// TIA Portal V17 program export: 1 tag tables, 23 data types, 8 data blocks, 12 code blocks (in call order from the OBs), 7 instance data blocks

VAR_GLOBAL   // PLC tag table "默认变量表"
   Tag_1 AT %M0.2 : Bool;
   System_Byte AT %MB1 : Byte;
   FirstScan AT %M1.0 : Bool;
   DiagStatusUpdate AT %M1.1 : Bool;
   AlwaysTRUE AT %M1.2 : Bool;
   AlwaysFALSE AT %M1.3 : Bool;
   Clock_Byte AT %MB0 : Byte;
   Clock_10Hz AT %M0.0 : Bool;
   Clock_5Hz AT %M0.1 : Bool;
   "Clock_2.5Hz" AT %M0.2 : Bool;
   Clock_2Hz AT %M0.3 : Bool;
   "Clock_1.25Hz" AT %M0.4 : Bool;
   Clock_1Hz AT %M0.5 : Bool;
   "Clock_0.625Hz" AT %M0.6 : Bool;
   "Clock_0.5Hz" AT %M0.7 : Bool;
   "PositioningAxis_1_Actor_Interface_AddressIn(8)" AT %I256.0 : "PD_TEL105_IN";
   "PositioningAxis_1_Actor_Interface_AddressOut(8)" AT %Q256.0 : "PD_TEL105_OUT";
   profiSafeCtrl1 AT %Q276.0 : "LDrvSafe_typeSinaTlg901Control";
   proSafeStatus1 AT %I276.0 : "LDrvSafe_typeSinaTlg901Status";
   profiSafeCtrl2 AT %Q310.0 : "LDrvSafe_typeSinaSTlg30Control";
   profiSafeStatus2 AT %I310.0 : "LDrvSafe_typeSinaSTlg30Status";
   "PositioningAxis_2_Actor_Interface_AddressIn(7)" AT %I290.0 : "PD_TEL105_IN";
   "PositioningAxis_2_Actor_Interface_AddressOut(7)" AT %Q290.0 : "PD_TEL105_OUT";
END_VAR

TYPE "LDrvSafe_typeSinaSTlg30Control"
TITLE = LDrvSafe_typeSinaSTlg30Control
// Failsafe user-defined data type for PROFIsafe telegram 30 to control the Safety Integrated Functions of SINAMICS S
// stored: IsFailsafeCompliant true
   STRUCT
      STO { ExternalWritable := 'False'} : Bool;   // Safety Function Safe Torque Off
      SS1 { ExternalWritable := 'False'} : Bool;   // Safety Function Safe Stop 1
      SS2 { ExternalWritable := 'False'} : Bool;   // Safety Function Safe Stop 2
      SOS { ExternalWritable := 'False'} : Bool;   // Safety Function Safe Operating Stop
      SLS { ExternalWritable := 'False'} : Bool;   // Safety Function Safely-limited Speed
      reserved1 { ExternalWritable := 'False'} : Bool;   // Reserve bit 1
      SLP { ExternalWritable := 'False'} : Bool;   // Safety Function Safely-limited Position
      internalEventAcknowledge { ExternalWritable := 'False'} : Bool;   // Acknowledge Safety errors in the drive
      SLA { ExternalWritable := 'False'} : Bool;   // Safety Function Safely-limited Acceleration
      selectSLSbit0 { ExternalWritable := 'False'} : Bool;   // Select one of the the four SLS limits; operates together with bit 1
      selectSLSbit1 { ExternalWritable := 'False'} : Bool;   // Select one of the the four SLS limits; operates together with bit 0
      reserved3 { ExternalWritable := 'False'} : Bool;   // Reserve bit 3
      SDIpositive { ExternalWritable := 'False'} : Bool;   // Safety Function Safe Direction (positive direction)
      SDInegative { ExternalWritable := 'False'} : Bool;   // Safety Function Safe Direction (negative direction)
      reserved4 { ExternalWritable := 'False'} : Bool;   // Reserve bit 4
      reserved5 { ExternalWritable := 'False'} : Bool;   // Reserve bit 5
   END_STRUCT;
END_TYPE

TYPE "LDrvSafe_typeSinaSTlg30Status"
TITLE = LDrvSafe_typeSinaSTlg30Status
// Failsafe user-defined data type for PROFIsafe telegram 30 to get status information of Safety Integrated Functions of SINAMICS S
// stored: IsFailsafeCompliant true
   STRUCT
      STOactive { ExternalWritable := 'False'} : Bool;   // Safety Function Safe Torque Off active
      SS1active { ExternalWritable := 'False'} : Bool;   // Safety Function Safe Stop 1 active
      SS2active { ExternalWritable := 'False'} : Bool;   // Safety Function Safe Stop 2 active
      SOSactive { ExternalWritable := 'False'} : Bool;   // Safety Function Safe Operating Stop active
      SLSactive { ExternalWritable := 'False'} : Bool;   // Safety Function Safely-limited Speed active
      reserved1 { ExternalWritable := 'False'} : Bool;   // Reserve bit 1
      SLPactive { ExternalWritable := 'False'} : Bool;   // Safety Function Safely-limited Position active
      internalEvent { ExternalWritable := 'False'} : Bool;   // Internal Event occured (Safety error in SINAMICS)
      SLAactive { ExternalWritable := 'False'} : Bool;   // Safety Function Safely-limited Acceleration active
      SLSbit0Active { ExternalWritable := 'False'} : Bool;   // One of the the four SLS limits is active; operates together with bit 1
      SLSbit1Active { ExternalWritable := 'False'} : Bool;   // One of the the four SLS limits is active; operates together with bit 0
      SOSselected { ExternalWritable := 'False'} : Bool;   // Safety Function Safe Operating Stop selected (not active yet)
      SDIpositiveActive { ExternalWritable := 'False'} : Bool;   // Safety Function Safe Direction (positive direction) active
      SDInegativeActive { ExternalWritable := 'False'} : Bool;   // Safety Function Safe Direction (negative direction) active
      reserved3 { ExternalWritable := 'False'} : Bool;   // Reserve bit 3
      SSMactive { ExternalWritable := 'False'} : Bool;   // Safety Function Safe Speed Monitor; signals, if safe speed is below paramterizable speed limit
   END_STRUCT;
END_TYPE

TYPE "LDrvSafe_typeSinaTlg901Control"
TITLE = LDrvSafe_typeSinaTlg901Control
// Failsafe user-defined data type for PROFIsafe telegram 901 to control the Safety Integrated Functions of SINAMICS
// stored: IsFailsafeCompliant true
   STRUCT
      STO { ExternalWritable := 'False'} : Bool;   // Safety Function Safe Torque Off
      SS1 { ExternalWritable := 'False'} : Bool;   // Safety Function Safe Stop 1
      SS2 { ExternalWritable := 'False'} : Bool;   // Safety Function Safe Stop 2
      SOS { ExternalWritable := 'False'} : Bool;   // Safety Function Safe Operating Stop
      SLS { ExternalWritable := 'False'} : Bool;   // Safety Function Safely-limited Speed
      reserved1 { ExternalWritable := 'False'} : Bool;   // Reserve bit 1
      SLP { ExternalWritable := 'False'} : Bool;   // Safety Function Safely-limited Position
      internalEventAcknowledge { ExternalWritable := 'False'} : Bool;   // Acknowledge Safety errors in the drive
      SLA { ExternalWritable := 'False'} : Bool;   // Safety Function Safely-limited Acceleration
      selectSLSbit0 { ExternalWritable := 'False'} : Bool;   // Select one of the the four SLS limits; operates together with bit 1
      selectSLSbit1 { ExternalWritable := 'False'} : Bool;   // Select one of the the four SLS limits; operates together with bit 0
      reserved2 { ExternalWritable := 'False'} : Bool;   // Reserve bit 2
      SDIpositive { ExternalWritable := 'False'} : Bool;   // Safety Function Safe Direction (positive direction)
      SDInegative { ExternalWritable := 'False'} : Bool;   // Safety Function Safe Direction (negative direction)
      reserved4 { ExternalWritable := 'False'} : Bool;   // Reserve bit 4
      reserved5 { ExternalWritable := 'False'} : Bool;   // Reserve bit 5
      reserved6 { ExternalWritable := 'False'} : Bool;   // Reserve bit 6
      reserved7 { ExternalWritable := 'False'} : Bool;   // Reserve bit 7
      reserved8 { ExternalWritable := 'False'} : Bool;   // Reserve bit 8
      selectSLPrange { ExternalWritable := 'False'} : Bool;   // Select one of the two SLP ranges
      reserved9 { ExternalWritable := 'False'} : Bool;   // Reserve bit 9
      reserved10 { ExternalWritable := 'False'} : Bool;   // Reserve bit 10
      reserved11 { ExternalWritable := 'False'} : Bool;   // Reserve bit 11
      SCA { ExternalWritable := 'False'} : Bool;   // Safety Function Safe Cam
      selectGearboxStageBit0 { ExternalWritable := 'False'} : Bool;   // Select one of the the eight gearbox stages; operates together with bit 1 and 2
      selectGearboxStageBit1 { ExternalWritable := 'False'} : Bool;   // Select one of the the eight gearbox stages; operates together with bit 0 and 2
      selectGearboxStageBit2 { ExternalWritable := 'False'} : Bool;   // Select one of the the eight gearbox stages; operates together with bit 0 and 1
      switchoverGearboxStage { ExternalWritable := 'False'} : Bool;   // Higher position tolerance at gearbox switching
      SS2E { ExternalWritable := 'False'} : Bool;   // Safety Function Safe Stop 2 with external stop
      reserved13 { ExternalWritable := 'False'} : Bool;   // Reserve bit 13
      reserved14 { ExternalWritable := 'False'} : Bool;   // Reserve bit 14
      reserved15 { ExternalWritable := 'False'} : Bool;   // Reserve bit 15
      variableSLS { ExternalWritable := 'False'} : Int;   // SLS limit 1 can be varied within 1 and 32.767 (0.03 and 100%)
   END_STRUCT;
END_TYPE

TYPE "LDrvSafe_typeSinaTlg901Status"
TITLE = LDrvSafe_typeSinaTlg901Status
// Failsafe user-defined data type for PROFIsafe telegram 901 to get status information of Safety Integrated Functions of SINAMICS
// stored: IsFailsafeCompliant true
   STRUCT
      STOactive { ExternalWritable := 'False'} : Bool;   // Safety Function Safe Torque Off active
      SS1active { ExternalWritable := 'False'} : Bool;   // Safety Function Safe Stop 1 active
      SS2active { ExternalWritable := 'False'} : Bool;   // Safety Function Safe Stop 2 active
      SOSactive { ExternalWritable := 'False'} : Bool;   // Safety Function Safe Operating Stop active
      SLSactive { ExternalWritable := 'False'} : Bool;   // Safety Function Safely-limited Speed active
      reserved1 { ExternalWritable := 'False'} : Bool;   // Reserve bit 1
      SLPactive { ExternalWritable := 'False'} : Bool;   // Safety Function Safely-limited Position active
      internalEvent { ExternalWritable := 'False'} : Bool;   // Internal Event occured (Safety error in SINAMICS)
      SLAactive { ExternalWritable := 'False'} : Bool;   // Safety Function Safely-limited Acceleration active
      SLSbit0Active { ExternalWritable := 'False'} : Bool;   // One of the the four SLS limits is active; operates together with bit 1
      SLSbit1Active { ExternalWritable := 'False'} : Bool;   // One of the the four SLS limits is active; operates together with bit 0
      reserved3 { ExternalWritable := 'False'} : Bool;   // Reserve bit 3
      SDIpositiveActive { ExternalWritable := 'False'} : Bool;   // Safety Function Safe Direction (positive direction) active
      SDInegativeActive { ExternalWritable := 'False'} : Bool;   // Safety Function Safe Direction (negative direction) active
      reserved4 { ExternalWritable := 'False'} : Bool;   // Reserve bit 4
      SSMactive { ExternalWritable := 'False'} : Bool;   // Safety Function Safe Speed Monitor; signals, if safe speed is below paramterizable speed limit
      reserved5 { ExternalWritable := 'False'} : Bool;   // Reserve bit 5
      reserved6 { ExternalWritable := 'False'} : Bool;   // Reserve bit 6
      reserved7 { ExternalWritable := 'False'} : Bool;   // Reserve bit 7
      SLPrangeActive { ExternalWritable := 'False'} : Bool;   // SLP position range 1 or 2 is active
      reserved8 { ExternalWritable := 'False'} : Bool;   // Reserve bit 8
      reserved9 { ExternalWritable := 'False'} : Bool;   // Reserve bit 9
      safePositionValid { ExternalWritable := 'False'} : Bool;   // Safe Position is valid
      safelyReferenced { ExternalWritable := 'False'} : Bool;   // Drive is safely referenced
      statusFDI0 { ExternalWritable := 'False'} : Bool;   // Status of Failsafe Digital Input 0
      statusFDI1 { ExternalWritable := 'False'} : Bool;   // Status of Failsafe Digital Input 1
      statusFDI2 { ExternalWritable := 'False'} : Bool;   // Status of Failsafe Digital Input 2
      reserved10 { ExternalWritable := 'False'} : Bool;   // Reserve bit 10
      SS2Eactive { ExternalWritable := 'False'} : Bool;   // Safety Function SS2E active
      SOSselected { ExternalWritable := 'False'} : Bool;   // Safety Function Safe Operating Stop selected (not active yet)
      SLPupperLimitMaintained { ExternalWritable := 'False'} : Bool;   // SLP: upper limit maintained
      SLPlowerLimitMaintained { ExternalWritable := 'False'} : Bool;   // SLP: lower limit maintained
      variableSLSvalue { ExternalWritable := 'False'} : Int;   // Actual SLS value for SLS limit 1
      cycleCounter { ExternalWritable := 'False'} : Int;   // Counter for the Safety cycle
      safePosition { ExternalWritable := 'False'} : Int;   // Current actual position value
   END_STRUCT;
END_TYPE

TYPE "typeFifo"
// stored: IsFailsafeCompliant false
   STRUCT
      enqueue : Bool;
      dequeue : Bool;
      reset : Bool;
      clear : Bool;
      initialItem : DInt;
      item : DInt;
      buffer : Array[0..9] of DInt;
   END_STRUCT;
END_TYPE

TYPE "typeFileReadWrite"
// stored: IsFailsafeCompliant false
   STRUCT
      start : Bool;
      offset : UDInt;
      length : UDInt;
      data : Array[0..999] of Byte;
      resultLength : UDInt;
      done : Bool;
      busy : Bool;
      status : Word;
      memErrStatus : Word;
   END_STRUCT;
END_TYPE

TYPE "LAxisCtrl_typeAxisConfig"
TITLE = LAxisCtrl_typeAxisConfig
// Support: tech.team.motioncontrol@siemens.com
// stored: IsFailsafeCompliant false
   STRUCT
      generalSettings : "LAxisCtrl_typeGeneralSettings";   // Configuration of general settings
      power : "LAxisCtrl_typePower";   // Configuration of MC_POWER function
      jog : "LAxisCtrl_typeJog";   // Configuration of JOG function
      moveVelocity : "LAxisCtrl_typeMoveVelocity";   // Configuration of MC_MOVEVELOCITY function
      stop : "LAxisCtrl_typeStop";   // Configuration of MC_HALT function
      fastStop : "LAxisCtrl_typeFastStop";   // Configuration of MC_HALT function (alternative dynamics)
      torqueLimiting : "LAxisCtrl_typeTorqueLimiting";   // Configuration of MC_TORQUELIMITING function
      homing : "LAxisCtrl_typeHoming";   // Configuration of HOMING function
      posRelative : "LAxisCtrl_typePosRelative";   // Configuration of MC_MOVERELATIVE function
      posAbsolute : "LAxisCtrl_typePosAbsolute";   // Configuration of MC_MOVEABSOLUTE function
      posSuperimposed : "LAxisCtrl_typePosSuperimposed";   // Configuration of MC_MOVESUPERIMPOSED function
      gearInRelative : "LAxisCtrl_typeGearInRelative";   // Configuration of MC_GEARIN function
      gearInAbsolute : "LAxisCtrl_typeGearInAbsolute";   // Configuration of MC_GEARIN_POS function
      camIn : "LAxisCtrl_typeCamIn";   // Configuration of MC_CAMIN function
      phasing : "LAxisCtrl_typePhasing";   // Configuration of MC_PHASING function
   END_STRUCT;
END_TYPE

TYPE "LAxisCtrl_typeDiagnostics"
TITLE = LAxisCtrl_typeDiagnostics
// Support: tech.team.motioncontrol@siemens.com
// stored: IsFailsafeCompliant false
   STRUCT
      status { ExternalWritable := 'False'} : Word := 16#0000;   // Status of FB when error occurred
      subfunctionStatus { ExternalWritable := 'False'} : Word := 16#0000;   // ErrorID of called subfunction
      basicMotionState { ExternalWritable := 'False'} : DInt := 0;   // Current basic motion state when error occurred
      superimposedMotionState { ExternalWritable := 'False'} : DInt := 0;   // Current superimposed motion state when error occurred
   END_STRUCT;
END_TYPE

TYPE "LAxisCtrl_typeCamIn"
TITLE = LAxisCtrl_typeCamIn
// Support: tech.team.motioncontrol@siemens.com
// stored: IsFailsafeCompliant false
   STRUCT
      masterOffset : LReal := 0.0;   // Offset of leading values of cam
      slaveOffset : LReal := 0.0;   // Offset of following values of cam
      masterScaling : LReal := 1.0;   // Scaling the leading values of the cam
      slaveScaling : LReal := 1.0;   // Scaling the following values of the cam
      masterSyncPosition : LReal := 0.0;   // Starting point in the cam/distance from the cam start with reference to the scaled cam
      syncProfileReference : DInt := 1;   // Synchronization profile (0: Sync. using dynamic parameters; 1: Sync. using leading value distance; 2: Direct sync. setting; 3: Subsequent sync. using leading value distance; 4: Subsequent sync. using leading value distance starting from current leading value position)
      masterStartDistance : LReal := 0.0;   // Leading value distance (when "SyncProfileReference" = 1)
      velocity : LReal := -1.0;   // Velocity for synchronization (when "SyncProfileReference" = 0; Value > 0.0: The specified value is used; Value = 0.0: Not permitted; Value < 0.0: Use of the default value configured in the technology object)
      acceleration : LReal := -1.0;   // Acceleration for synchronization (when "SyncProfileReference" = 0; Value > 0.0: The specified value is used; Value = 0.0: Not permitted; Value < 0.0: Use of the default value configured in the technology object)
      deceleration : LReal := -1.0;   // Deceleration for synchronization (when "SyncProfileReference" = 0; Value > 0.0: The specified value is used; Value = 0.0: Not permitted; Value < 0.0: Use of the default value configured in the technology object)
      jerk : LReal := -1.0;   // Jerk for synchronization (when "SyncProfileReference" = 0; Value > 0.0: Smooth velocity profile, the specified value is used; Value = 0.0: Trapezoid velocity profile; Value < 0.0: Use of the default value configured in the technology object)
      applicationMode : DInt := 0;   // Application of the cam (0: Once/not cyclic; 1: Cyclic ; 2: Cyclic appending)
      syncDirection : DInt := 1;   // Direction for synchronization only in effect for axes with activated modulo setting (1: Forward direction; 2: Backward direction; 3: Shortest way)
   END_STRUCT;
END_TYPE

TYPE "LAxisCtrl_typeFastStop"
TITLE = LAxisCtrl_typeFastStop
// Support: tech.team.motioncontrol@siemens.com
// stored: IsFailsafeCompliant false
   STRUCT
      deceleration : LReal := -1.0;   // Deceleration for fast stop (Value > 0.0: The specified value is used; Value <= 0.0: emergency deceleration of the technology object is used)
      jerk : LReal := -1.0;   // Jerk for fast stop (Value > 0.0: Smooth velocity profile, the specified value is used; Value = 0.0: Trapezoid velocity profile; Value < 0.0: Use of the default value configured in the technology object)
      abortAcceleration : Bool := FALSE;   // TRUE: The acceleration is set to 0.0 at the start of the job, and the deceleration immediately builds up; FALSE: The current acceleration at the start of the job is reduced using the configured jerk. Afterwards, the deceleration builds up
      replaceStopPossible : Bool := FALSE;   // TRUE: Fast stop command can be replaced by another command
   END_STRUCT;
END_TYPE

TYPE "LAxisCtrl_typeGearInAbsolute"
TITLE = LAxisCtrl_typeGearInAbsolute
// Support: tech.team.motioncontrol@siemens.com
// stored: IsFailsafeCompliant false
   STRUCT
      ratioNumerator : DInt := 1;   // Gear ratio numerator
      ratioDenominator : DInt := 1;   // Gear ratio denominator
      masterSyncPosition : LReal := 0.0;   // Synchronous position of leading axis
      slaveSyncPosition : LReal := 0.0;   // Synchronous position of following axis
      syncProfileReference : DInt := 1;   // Type of synchronization (0: Sync. using dynamic parameters; 1: Sync. using leading value distance; 3: Subsequent sync. using leading value distance)
      masterStartDistance : LReal := 0.0;   // Leading value distance (when "SyncProfileReference" = 1)
      velocity : LReal := -1.0;   // Velocity for synchronization (when "SyncProfileReference" = 0; Value > 0.0: The specified value is used; Value = 0.0: Not permitted; Value < 0.0: Use of the default value configured in the technology object)
      acceleration : LReal := -1.0;   // Acceleration for synchronization (when "SyncProfileReference" = 0; Value > 0.0: The specified value is used; Value = 0.0: Not permitted; Value < 0.0: Use of the default value configured in the technology object)
      deceleration : LReal := -1.0;   // Deceleration for synchronization (when "SyncProfileReference" = 0; Value > 0.0: The specified value is used; Value = 0.0: Not permitted; Value < 0.0: Use of the default value configured in the technology object)
      jerk : LReal := -1.0;   // Jerk for synchronization (when "SyncProfileReference" = 0; Value > 0.0: Smooth velocity profile, the specified value is used; Value = 0.0: Trapezoid velocity profile; Value < 0.0: Use of the default value configured in the technology object)
      syncDirection : DInt := 1;   // Direction for synchronization only in effect for axes with activated modulo setting (1: Forward direction; 2: Backward direction; 3: Shortest way)
      ratioChangeOnTheFly : Bool := FALSE;   // TRUE: Changing gear ratio on-the-fly; FALSE: Ratio change requires a new rising edge at gearInAbsolute input
   END_STRUCT;
END_TYPE

TYPE "LAxisCtrl_typeGearInRelative"
TITLE = LAxisCtrl_typeGearInRelative
// Support: tech.team.motioncontrol@siemens.com
// stored: IsFailsafeCompliant false
   STRUCT
      ratioNumerator : DInt := 1;   // Gear ratio numerator
      ratioDenominator : DInt := 1;   // Gear ratio denominator
      acceleration : LReal := -1.0;   // Acceleration for synchronization (when "SyncProfileReference" = 0; Value > 0.0: The specified value is used; Value = 0.0: Not permitted; Value < 0.0: Use of the default value configured in the technology object)
      deceleration : LReal := -1.0;   // Deceleration for synchronization (when "SyncProfileReference" = 0; Value > 0.0: The specified value is used; Value = 0.0: Not permitted; Value < 0.0: Use of the default value configured in the technology object)
      jerk : LReal := -1.0;   // Jerk for synchronization (when "SyncProfileReference" = 0; Value > 0.0: Smooth velocity profile, the specified value is used; Value = 0.0: Trapezoid velocity profile; Value < 0.0: Use of the default value configured in the technology object)
      ratioChangeOnTheFly : Bool := FALSE;   // TRUE: Changing gear ratio on-the-fly; FALSE: Ratio change requires a new rising edge at gearInRelative input
   END_STRUCT;
END_TYPE

TYPE "LAxisCtrl_typeGeneralSettings"
TITLE = LAxisCtrl_typeGeneralSettings
// Support: tech.team.motioncontrol@siemens.com
// stored: IsFailsafeCompliant false
   STRUCT
      stopOnError : Bool := TRUE;   // TRUE: In case of error the axis will be stopped automatically with fastStop dynamics
      resetWithRestart : Bool := FALSE;   // TRUE: Reinitialization of the technology object and acknowledgment of pending technology alarms. The technology object is reinitialized with the configured start values; FALSE: Acknowledgment of queued technology alarms
      abortWaitingSyncCmd : Bool := TRUE;   // TRUE: Abort waiting synchronous command in case of new basic motion command automatically
   END_STRUCT;
END_TYPE

TYPE "LAxisCtrl_typeHoming"
TITLE = LAxisCtrl_typeHoming
// Support: tech.team.motioncontrol@siemens.com
// stored: IsFailsafeCompliant false
   STRUCT
      position : LReal := 0.0;   // The specified value is used according to the selected "Mode"
      mode : Int := 0;   // Operation mode; 0: Direct homing (absolute); 1: Direct homing (relative); 2: Passive homing (without reset); 3: Active homing; 5: Active homing (Position parameter has no effect); 6: Absolute encoder adjustment (relative); 7: Absolute encoder adjustment (absolute); 8:Passive homing ; 9: Abort passive homing; 10: Passive homing (Position parameter has no effect); 11: Set setpoint position (absolute); 12: Shift the setpoint position (relative)
      extendedMode : DInt := -1;   // -1: No extended homing mode (parameter "mode" is effective); 0: Homing on fixed stop; 1: Homing on fixed stop with moving out of clamping
      extendedModeTorqueLimit : LReal := 0.0;   // Value of the torque/force for extended homing mode
   END_STRUCT;
END_TYPE

TYPE "LAxisCtrl_typeJog"
TITLE = LAxisCtrl_typeJog
// Support: tech.team.motioncontrol@siemens.com
// stored: IsFailsafeCompliant false
   STRUCT
      velocity : LReal := 0.0;   // Velocity for jogging (Value > 0.0: The specified value is used; Value = 0.0: Permitted; Value < 0.0: The absolute value of the specified value is used)
      acceleration : LReal := -1.0;   // Acceleration for jogging (Value > 0.0: The specified value is used; Value = 0.0: Not permitted; Value < 0.0: Use of the default value configured in the technology object)
      deceleration : LReal := -1.0;   // Deceleration for jogging (Value > 0.0: The specified value is used; Value = 0.0: Not permitted; Value < 0.0: Use of the default value configured in the technology object)
      jerk : LReal := -1.0;   // Jerk for jogging (Value > 0.0: Smooth velocity profile, the specified value is used; Value = 0.0: Trapezoid velocity profile; Value < 0.0: Use of the default value configured in the technology object)
      positionControlled : Bool := TRUE;   // TRUE: Position-controlled mode; FALSE: Non position-controlled operation
      increment : LReal := 0.0;   // Increment/distance for incremental jogging
      mode : DInt := 0;   // 0: Continuous jogging; 1: Incremental jogging new increment (starts with new increment); 2: Incremental jogging continue increment (continue the last increment if not completed)
   END_STRUCT;
END_TYPE

TYPE "LAxisCtrl_typeMoveVelocity"
TITLE = LAxisCtrl_typeMoveVelocity
// Support: tech.team.motioncontrol@siemens.com
// stored: IsFailsafeCompliant false
   STRUCT
      velocity : LReal := 0.0;   // Velocity/Speed for motion process (Value = 0.0: Permitted)
      acceleration : LReal := -1.0;   // Acceleration setpoint for motion process (Value > 0.0: The specified value is used; Value = 0.0: Not permitted; Value < 0.0: Use of the default value configured in the technology object)
      deceleration : LReal := -1.0;   // Deceleration setpoint for motion process (Value > 0.0: The specified value is used; Value = 0.0: Not permitted; Value < 0.0: Use of the default value configured in the technology object)
      jerk : LReal := -1.0;   // Jerk for velocity specification (Value > 0.0: Smooth velocity profile, the specified value is used; (Value = 0.0: Trapezoid velocity profile; (Value < 0.0: Use of the default value configured in the technology object)
      direction : Int := 0;   // Motion direction of the axis (0: The sign of the velocity parameter defines the direction; 1: Positive direction; 2: Negative direction)
      positionControlled : Bool := TRUE;   // TRUE: Position-controlled operation; FALSE: Non position-controlled operation
      velocityChangeOnTheFly : Bool := FALSE;   // TRUE: Changing velocity on-the-fly; FALSE: Velocity change requires a new rising edge on moveVelocity input
   END_STRUCT;
END_TYPE

TYPE "LAxisCtrl_typePhasing"
TITLE = LAxisCtrl_typePhasing
// Support: tech.team.motioncontrol@siemens.com
// stored: IsFailsafeCompliant false
   STRUCT
      phaseShift : LReal := 0.0;   // Absolute or relative leading value shift
      velocity : LReal := -1.0;   // Velocity for leading value shift, added to synchronous operation motion (Value > 0.0: The specified value is used; Value = 0.0: Not permitted; Value < 0.0: Use of the default value configured in the technology object)
      acceleration : LReal := -1.0;   // Acceleration for leading value shift, added to synchronous operation motion (Value > 0.0: The specified value is used; Value = 0.0: Not permitted; Value < 0.0: Use of the default value configured in the technology object)
      deceleration : LReal := -1.0;   // Deceleration for leading value shift, added to synchronous operation motion (Value > 0.0: The specified value is used; Value = 0.0: Not permitted; Value < 0.0: Use of the default value configured in the technology object)
      jerk : LReal := -1.0;   // Jerk for leading value shift, added to synchronous operation motion (Value > 0.0: Smooth velocity profile, the specified value is used; Value = 0.0: Trapezoid velocity profile; Value < 0.0: Use of the default value configured in the technology object)
      phaseAbsolute : Bool := TRUE;   // Indicates the type of phase shift. TRUE: Shift the leading value as an absolute shift; FALSE: Shift the leading value relative to the existing leading value shift
      phaseShiftChangeOnTheFly : Bool := FALSE;   // TRUE: Changing phase shift on-the-fly at absolute phasing; FALSE: Phase shift change requires a new rising edge at phasing input
   END_STRUCT;
END_TYPE

TYPE "LAxisCtrl_typePosAbsolute"
TITLE = LAxisCtrl_typePosAbsolute
// Support: tech.team.motioncontrol@siemens.com
// stored: IsFailsafeCompliant false
   STRUCT
      position : LReal := 0.0;   // Absolute target position
      velocity : LReal := -1.0;   // Velocity setpoint for absolute positioning (Value > 0.0: The specified value is used; Value = 0.0: Not permitted; Value < 0.0: Use of the default value configured in the technology object)
      acceleration : LReal := -1.0;   // Acceleration setpoint for absolute positioning (Value > 0.0: The specified value is used; Value = 0.0: Not permitted; Value < 0.0: Use of the default value configured in the technology object)
      deceleration : LReal := -1.0;   // Deceleration setpoint for absolute positioning (Value > 0.0: The specified value is used; Value = 0.0: Not permitted; Value < 0.0: Use of the default value configured in the technology object)
      jerk : LReal := -1.0;   // Jerk for absolute positioning (Value > 0.0: Smooth velocity profile, the specified value is used; (Value = 0.0: Trapezoid velocity profile; (Value < 0.0: Use of the default value configured in the technology object)
      direction : Int := 1;   // Motion direction of the axis (1: Positive direction; 2: Negative direction; 3: Shortest way)
      positionChangeOnTheFly : Bool := FALSE;   // TRUE: Changing position on-the-fly; FALSE: Position change requires a new rising edge at posAbsolute input
      velocityChangeOnTheFly : Bool := FALSE;   // TRUE: Changing velocity on-the-fly; FALSE: Velocity change requires a new rising edge at posAbsolute input
   END_STRUCT;
END_TYPE

TYPE "LAxisCtrl_typePosRelative"
TITLE = LAxisCtrl_typePosRelative
// Support: tech.team.motioncontrol@siemens.com
// stored: IsFailsafeCompliant false
   STRUCT
      distance : LReal := 0.0;   // Distance for positioning process
      velocity : LReal := -1.0;   // Velocity setpoint for relative positioning (Value > 0.0: The specified value is used; Value = 0.0: Not permitted; Value < 0.0: Use of the default value configured in the technology object)
      acceleration : LReal := -1.0;   // Acceleration setpoint for relative positioning (Value > 0.0: The specified value is used; Value = 0.0: Not permitted; Value < 0.0: Use of the default value configured in the technology object)
      deceleration : LReal := -1.0;   // Deceleration setpoint for relative positioning (Value > 0.0: The specified value is used; Value = 0.0: Not permitted; Value < 0.0: Use of the default value configured in the technology object)
      jerk : LReal := -1.0;   // Jerk for relative positioning (Value > 0.0: Smooth velocity profile, the specified value is used; Value = 0.0: Trapezoid velocity profile; Value < 0.0: Use of the default value configured in the technology object)
      direction : DInt := 0;   // Motion direction of the axis (0: The sign of the distance parameter defines the direction; 1: Positive direction; 2: Negative direction)
   END_STRUCT;
END_TYPE

TYPE "LAxisCtrl_typePosSuperimposed"
TITLE = LAxisCtrl_typePosSuperimposed
// Support: tech.team.motioncontrol@siemens.com
// stored: IsFailsafeCompliant false
   STRUCT
      distance : LReal := 0.0;   // Distance for superimposed positioning
      velocityDiff : LReal := -1.0;   // Maximum velocity deviation compared to the active motion (Value > 0.0: The specified value is used; Value = 0.0: Not permitted; Value < 0.0: Use of the default value configured in the technology object)
      acceleration : LReal := -1.0;   // Acceleration for positioning (Value > 0.0: The specified value is used; Value = 0.0: Not permitted; Value < 0.0: Use of the default value configured in the technology object)
      deceleration : LReal := -1.0;   // Deceleration for positioning (Value > 0.0: The specified value is used; Value = 0.0: Not permitted; Value < 0.0: Use of the default value configured in the technology object)
      jerk : LReal := -1.0;   // Jerk for positioning (Value > 0.0: Smooth velocity profile, the specified value is used; Value = 0.0: Trapezoid velocity profile; Value < 0.0: Use of the default value configured in the technology object)
      direction : DInt := 0;   // Motion direction of the axis (0: The sign of the distance parameter defines the direction; 1: Positive negative; 2: Negative direction)
   END_STRUCT;
END_TYPE

TYPE "LAxisCtrl_typePower"
TITLE = LAxisCtrl_typePower
// Support: tech.team.motioncontrol@siemens.com
// stored: IsFailsafeCompliant false
   STRUCT
      startMode : DInt := 1;   // 0: Enable axis not position-controlled; 1: Enable axis position-controlled (This parameter is ignored when a speed axis or external encoder is used)
      stopMode : Int := 0;   // 0: Emergency stop; 1: Immediate stop; 2: Stop with maximum dynamic values
      syncMotionSimulation : Bool := FALSE;   // TRUE: Start the simulation of synchronous operation automatically with falling edge at enableAxis; FALSE: No simulation of synchronous operation
   END_STRUCT;
END_TYPE

TYPE "LAxisCtrl_typeStop"
TITLE = LAxisCtrl_typeStop
// Support: tech.team.motioncontrol@siemens.com
// stored: IsFailsafeCompliant false
   STRUCT
      deceleration : LReal := -1.0;   // Deceleration setpoint for stop (Value > 0.0: The specified value is used; Value = 0.0: Not permitted; Value < 0.0: Use of the default value configured in the technology object)
      jerk : LReal := -1.0;   // Jerk for stop (Value > 0.0: Smooth velocity profile, the specified value is used; Value = 0.0: Trapezoid velocity profile; Value < 0.0: Use of the default value configured in the technology object)
      abortAcceleration : Bool := FALSE;   // TRUE: The acceleration is set to 0.0 at the start of the job, and the deceleration immediately builds up; FALSE: The current acceleration at the start of the job is reduced using the configured jerk. Afterwards, the deceleration builds up
   END_STRUCT;
END_TYPE

TYPE "LAxisCtrl_typeTorqueLimiting"
TITLE = LAxisCtrl_typeTorqueLimiting
// Support: tech.team.motioncontrol@siemens.com
// stored: IsFailsafeCompliant false
   STRUCT
      limit : LReal := -1.0;   // Value of force/torque limiting (in the configured unit of measurement)
      mode : DInt := 0;   // 0: Force/Torque limiting; 1: Fixed stop detection
   END_STRUCT;
END_TYPE

DATA_BLOCK "DataFromSafety"   // DB6
{ S7_Optimized_Access := 'TRUE' }
VERSION : 0.1
// stored: AutoNumber true, DBAccessibleFromOPCUA true, DBAccessibleFromWebserver true, IsOnlyStoredInLoadMemory false, IsRetainMemResEnabled false, IsWriteProtectedInAS false, MemoryReserve 100
   VAR
      ss1ActiveAxis1 : Bool;
      ss1ActiveAxis2 : Bool;
   END_VAR
BEGIN
END_DATA_BLOCK

DATA_BLOCK "StringDb"   // DB10
{ S7_Optimized_Access := 'FALSE' }
VERSION : 0.1
// stored: AutoNumber true, DBAccessibleFromOPCUA true, DBAccessibleFromWebserver true, IsOnlyStoredInLoadMemory false, IsWriteProtectedInAS false
   VAR
      name1 : String;
      testBool : Bool;
   END_VAR
BEGIN
END_DATA_BLOCK

DATA_BLOCK "Test"   // DB4
{ S7_Optimized_Access := 'TRUE' }
VERSION : 0.1
// stored: AutoNumber true, DBAccessibleFromOPCUA true, DBAccessibleFromWebserver true, IsOnlyStoredInLoadMemory false, IsRetainMemResEnabled false, IsWriteProtectedInAS false, MemoryReserve 100
   VAR
      stoAxis1 : Bool := 1;
      stoAxis2 : Bool := 1;
      ss1Axis1 : Bool := 1;
      reset : Bool;
      reintegration : Bool;
      ss1Axis2 : Bool := 1;
      enableAxis1 : Bool;
      enableAxis2 : Bool;
      moveVelocityAxis1 : Bool;
      moveVelocityAxis2 : Bool;
      homeAxis1 : Bool;
      configAxis1 : "LAxisCtrl_typeAxisConfig";
      configAxis2 { S7_SetPoint := 'True'} : "LAxisCtrl_typeAxisConfig";
      "jog+" { S7_SetPoint := 'True'} : Bool;
      "jog-" : Bool;
      stop : Bool;
      sto1 : Bool := 1;
      sto2 : Bool := 1;
      ss2Axis1 : Bool := 1;
      ss2Axis2 : Bool := 1;
      test : Bool := 0;
      fifo : "typeFifo";
      "name" { S7_SetPoint := 'True'} : Array[0..50] of String;
      name1 : String;
      "real" : Real;
      releaseEstop : Bool := true;
      releaseGate : Bool := true;
      enableMode : Bool := 0;
      stoActiveAxis1 : Bool;
      stoActiveAxis2 : Bool;
      ss1ActiveAxis1 : Bool;
      ss1ActiveAxis2 : Bool;
      ss2ActiveAxis1 : Bool;
      ss2ActiveAxis2 : Bool;
      slsActiveAxis1 : Bool;
      slsActiveAxis2 : Bool;
   END_VAR
BEGIN
   configAxis1.moveVelocity.velocity := 40.0;
   configAxis2.moveVelocity.velocity := 40.0;
END_DATA_BLOCK

DATA_BLOCK "TestSclDb"   // DB7
{ S7_Optimized_Access := 'TRUE' }
VERSION : 0.1
// stored: AutoNumber true, DBAccessibleFromOPCUA true, DBAccessibleFromWebserver true, IsOnlyStoredInLoadMemory false, IsRetainMemResEnabled false, IsWriteProtectedInAS false, MemoryReserve 100
   VAR
      start : Bool;
      state1 : Bool;
      state2 : Bool;
      state3 : Bool;
      state4 : Bool;
      state5 : Bool;
      state6 : Bool;
      nextStep : Bool;
      cond1 : Int;
      testCond1 : Bool;
      result : Bool;
      aArray : Array[0..9] of Int;
      bArray : Array[0..9] of Int;
      count : SInt := 9;
      string1 : Array[0..10] of String[50];
      string2 : Array[0..10] of String[50];
      string3 : Array[0..10] of String[50];
      dumpString : String;
   END_VAR
BEGIN
   bArray[0] := 1;
END_DATA_BLOCK

DATA_BLOCK "dataHandling111"   // DB2
{ S7_Optimized_Access := 'FALSE' }
VERSION : 0.1
// stored: AutoNumber true, DBAccessibleFromOPCUA true, DBAccessibleFromWebserver true, IsOnlyStoredInLoadMemory false, IsWriteProtectedInAS false
   VAR
      data : Array[0..3] of Byte;
   END_VAR
BEGIN
END_DATA_BLOCK

DATA_BLOCK "Data"   // DB147
{ S7_Optimized_Access := 'TRUE' }
VERSION : 0.1
// stored: AutoNumber true, DBAccessibleFromOPCUA true, DBAccessibleFromWebserver true, IsOnlyStoredInLoadMemory false, IsRetainMemResEnabled false, IsWriteProtectedInAS false, MemoryReserve 100
   VAR
      rdSysT { ExternalWritable := 'False'} : Struct
         retVal { ExternalWritable := 'False'} : Int;   // return value
         "time" { ExternalWritable := 'False'} : DTL;   // system time
      END_STRUCT;
      simulation : Struct
         amplitude : Real := 6.0;   // Amplitude
         offset : Real := -22.0;   // Offset
         periode : UDInt := 60000;   // Periode in milliseconds
         value { ExternalWritable := 'False'} : Real;   // Calculated Sinus value / Calculated Sinus values
      END_STRUCT;
   END_VAR
   VAR RETAIN
      write : Bool;   // trigger for data logging
      dataLogSameFile : Struct
         enable : Bool := TRUE;   // TRUE: enable function block
         delete : Bool;   // TRUE: Delete data log(s)
         data : Struct   // data logging data
            temperature : Real;   // temperature to log
            Pressure : Real;
            Flow : Real;
         END_STRUCT;
         done { ExternalWritable := 'False'} : Bool;   // TRUE: Commanded functionality has been completed successfully
         error { ExternalWritable := 'False'} : Bool;   // TRUE: An error occurred during the execution of the FB
         status { ExternalWritable := 'False'} : Word;   // Status of the FB "DataLog1x00"
         subFunctionStatus { ExternalWritable := 'False'} : Word;   // Subfunction status
         numberRecords { ExternalWritable := 'False'} : UDInt;   // Current number of data records in the data log
         sync { ExternalWritable := 'False'} : Bool;   // "numberRecords" is synchronized
         last { ExternalWritable := 'False'} : Struct
            done { ExternalWritable := 'False'} : Struct
               old { ExternalAccessible := 'False'; ExternalVisible := 'False'; ExternalWritable := 'False'} : Bool;   // Old value for edge detection
               "time" { ExternalWritable := 'False'} : DTL;   // last time of successful completion
            END_STRUCT;
            error { ExternalWritable := 'False'} : Struct
               old { ExternalAccessible := 'False'; ExternalVisible := 'False'; ExternalWritable := 'False'} : Bool;   // Old value for edge detection
               "time" { ExternalWritable := 'False'} : DTL;   // last time of completion with error
               status { ExternalWritable := 'False'} : Word;   // 16#8601: DataLogCreate, 16#8602: DataLogOpen, 16#8603: DataLogWrite, 16#8604: DataLogClear, 16#8605: DataLogClose, 16#8606: DataLogNewFile, 16#8607: DataLogDelete
               subFunctionStatus { ExternalWritable := 'False'} : Word;   // Subfunction status
            END_STRUCT;
         END_STRUCT;
      END_STRUCT;
      tmailcAlarm : Struct
         enable : Bool := TRUE;   // TRUE: enable function block
         toS : String[240] := 'receiver@siemens.de';   // Recipient address
         mailAddrParam : TMail_QDN_SEC;   // addressing parameters
         done { ExternalWritable := 'False'} : Bool;   // E-mail has been sent
         error { ExternalWritable := 'False'} : Bool;   // Error while sending the e-mail
         status { ExternalWritable := 'False'} : Word;   // Status when error occured
         last { ExternalWritable := 'False'} : Struct
            done { ExternalWritable := 'False'} : Struct
               old { ExternalAccessible := 'False'; ExternalVisible := 'False'; ExternalWritable := 'False'} : Bool;   // Old value for edge detection
               "time" { ExternalWritable := 'False'} : DTL;   // last time of successful completion
            END_STRUCT;
            error { ExternalWritable := 'False'} : Struct
               old { ExternalAccessible := 'False'; ExternalVisible := 'False'; ExternalWritable := 'False'} : Bool;   // Old value for edge detection
               "time" { ExternalWritable := 'False'} : DTL;   // last time of completion with error
               status { ExternalWritable := 'False'} : Word;   // Status when error occured
               sfbStatus { ExternalWritable := 'False'} : Word;   // Error related SFB status
            END_STRUCT;
         END_STRUCT;
      END_STRUCT;
      dataLogNewFile : Struct
         enable : Bool := TRUE;   // TRUE: enable function block
         delete : Bool;   // TRUE: Delete data log(s)
         data : Struct   // data logging data
            temperature : Real;   // temperature to log
            Pressure : Real;
            Flow : Real;
         END_STRUCT;
         done { ExternalWritable := 'False'} : Bool;   // TRUE: Commanded functionality has been completed successfully
         error { ExternalWritable := 'False'} : Bool;   // TRUE: An error occurred during the execution of the FB
         status { ExternalWritable := 'False'} : Word;   // Status of the FB "DataLog1x00"
         subFunctionStatus { ExternalWritable := 'False'} : Word;   // Subfunction status
         id { ExternalWritable := 'False'} : DWord;   // Object ID of the data log
         numberRecords { ExternalWritable := 'False'} : UDInt;   // Current number of data records in the data log
         sync { ExternalWritable := 'False'} : Bool;   // "numberRecords" is synchronized
         full { ExternalWritable := 'False'} : Bool;   // The maximum number of data records is reached
         fullOld { ExternalWritable := 'False'} : Bool;   // Old value for edge detection
         currentName { ExternalWritable := 'False'} : String;   // Current data log file name
         last { ExternalWritable := 'False'} : Struct
            done { ExternalWritable := 'False'} : Struct
               old { ExternalAccessible := 'False'; ExternalVisible := 'False'; ExternalWritable := 'False'} : Bool;   // Old value for edge detection
               "time" { ExternalWritable := 'False'} : DTL;   // last time of successful completion
            END_STRUCT;
            error { ExternalWritable := 'False'} : Struct
               old { ExternalAccessible := 'False'; ExternalVisible := 'False'; ExternalWritable := 'False'} : Bool;   // Old value for edge detection
               "time" { ExternalWritable := 'False'} : DTL;   // last time of completion with error
               status { ExternalWritable := 'False'} : Word;   // 16#8601: DataLogCreate, 16#8602: DataLogOpen, 16#8603: DataLogWrite, 16#8604: DataLogClear, 16#8605: DataLogClose, 16#8606: DataLogNewFile, 16#8607: DataLogDelete
               subFunctionStatus { ExternalWritable := 'False'} : Word;   // Subfunction status
            END_STRUCT;
         END_STRUCT;
      END_STRUCT;
      tmailcCsvTransfer : Struct
         enable : Bool := TRUE;   // TRUE: enable function block
         toS : String[240] := 'receiver@siemens.de';   // Recipient address
         mailAddrParam : TMail_QDN_SEC;   // addressing parameters
         attachment : TMail_FileReference;   // Attachment
         done { ExternalWritable := 'False'} : Bool;   // E-mail has been sent
         error { ExternalWritable := 'False'} : Bool;   // Error while sending the e-mail
         status { ExternalWritable := 'False'} : Word;   // Status when error occured
         last { ExternalWritable := 'False'} : Struct
            done { ExternalWritable := 'False'} : Struct
               old { ExternalAccessible := 'False'; ExternalVisible := 'False'; ExternalWritable := 'False'} : Bool;   // Old value for edge detection
               "time" { ExternalWritable := 'False'} : DTL;   // last time of successful completion
            END_STRUCT;
            error { ExternalWritable := 'False'} : Struct
               old { ExternalAccessible := 'False'; ExternalVisible := 'False'; ExternalWritable := 'False'} : Bool;   // Old value for edge detection
               "time" { ExternalWritable := 'False'} : DTL;   // last time of completion with error
               status { ExternalWritable := 'False'} : Word;   // Status when error occured
               sfbStatus { ExternalWritable := 'False'} : Word;   // Error related SFB status
            END_STRUCT;
         END_STRUCT;
      END_STRUCT;
   END_VAR
BEGIN
   tmailcAlarm.mailAddrParam.InterfaceId := 64;
   tmailcAlarm.mailAddrParam.ID := 1;
   tmailcAlarm.mailAddrParam.ConnectionType := 16#22;
   tmailcAlarm.mailAddrParam.WatchDogTime := T#60s;
   tmailcAlarm.mailAddrParam.MailServerQDN := 'smtp.gmail.com.';
   tmailcAlarm.mailAddrParam.UserName := 'sender@googlemail.com';
   tmailcAlarm.mailAddrParam.PassWord := 'Password';
   tmailcAlarm.mailAddrParam.From.LocalPartPlusAtSign := 'sender@';
   tmailcAlarm.mailAddrParam.From.FullQualifiedDomainName := 'googlemail.com';
   tmailcAlarm.mailAddrParam.RemotePort := 587;
   tmailcAlarm.mailAddrParam.ActivateSecureConn := true;
   tmailcAlarm.mailAddrParam.TLSServerCertRef := 43;
   tmailcCsvTransfer.mailAddrParam.InterfaceId := 64;
   tmailcCsvTransfer.mailAddrParam.ID := 2;
   tmailcCsvTransfer.mailAddrParam.ConnectionType := 16#22;
   tmailcCsvTransfer.mailAddrParam.WatchDogTime := T#60s;
   tmailcCsvTransfer.mailAddrParam.MailServerQDN := 'smtp.gmail.com.';
   tmailcCsvTransfer.mailAddrParam.UserName := 'sender@googlemail.com';
   tmailcCsvTransfer.mailAddrParam.PassWord := 'Password';
   tmailcCsvTransfer.mailAddrParam.From.LocalPartPlusAtSign := 'sender@';
   tmailcCsvTransfer.mailAddrParam.From.FullQualifiedDomainName := 'googlemail.com';
   tmailcCsvTransfer.mailAddrParam.RemotePort := 587;
   tmailcCsvTransfer.mailAddrParam.ActivateSecureConn := true;
   tmailcCsvTransfer.mailAddrParam.TLSServerCertRef := 43;
   tmailcCsvTransfer.attachment.DirectoryPath := '/DataLogs/';
   tmailcCsvTransfer.attachment.FileName := 'datalog.csv';
END_DATA_BLOCK

DATA_BLOCK "TestDataLog"   // DB12
{ S7_Optimized_Access := 'TRUE' }
VERSION : 0.1
// stored: AutoNumber true, DBAccessibleFromOPCUA true, DBAccessibleFromWebserver true, IsOnlyStoredInLoadMemory false, IsRetainMemResEnabled false, IsWriteProtectedInAS false, MemoryReserve 100
   VAR
      tag : Bool;
   END_VAR
BEGIN
END_DATA_BLOCK

DATA_BLOCK "SLI_gDB_FileHandling"   // DB11
{ S7_Optimized_Access := 'FALSE' }
VERSION : 0.1
// stored: AutoNumber true, DBAccessibleFromOPCUA true, DBAccessibleFromWebserver true, IsOnlyStoredInLoadMemory false, IsWriteProtectedInAS false
   VAR
      "name" : String := 'UserFiles/SLI_text.txt';
      fileWrite : "typeFileReadWrite";
      fileRead { S7_SetPoint := 'True'} : "typeFileReadWrite";
      fileDelete { S7_SetPoint := 'True'} : "typeFileReadWrite";
      data2 { S7_SetPoint := 'True'} : Array[0..999] of Byte;
   END_VAR
BEGIN
   fileWrite.length := 1000;
   fileWrite.data[0] := 16#10;
   fileWrite.data[1] := 11;
   fileWrite.data[2] := 12;
   fileWrite.data[3] := 13;
   fileWrite.data[4] := 14;
   fileWrite.data[5] := 15;
   fileWrite.data[6] := 16;
   fileWrite.data[7] := 17;
   fileWrite.data[8] := 18;
   fileWrite.data[9] := 19;
   fileWrite.data[10] := 20;
   data2[0] := 16#1;
   data2[1] := 2;
   data2[2] := 3;
   data2[3] := 4;
   data2[4] := 5;
   data2[5] := 6;
   data2[6] := 7;
   data2[7] := 8;
   data2[8] := 9;
   data2[9] := 10;
   data2[104] := 100;
END_DATA_BLOCK

ORGANIZATION_BLOCK "Main"   // OB1, LAD, ProgramCycle
TITLE = "Main Program Sweep (Cycle)"
{ S7_Optimized_Access := 'TRUE' }
VERSION : 0.1
// stored: AutoNumber true, IsIECCheckEnabled false, SetENOAutomatically false
   VAR_INPUT
      Initial_Call : Bool;   // Initial call of this OB
      Remanence : Bool;   // =True, if remanent data are available
   END_VAR
BEGIN

REGION Network 2
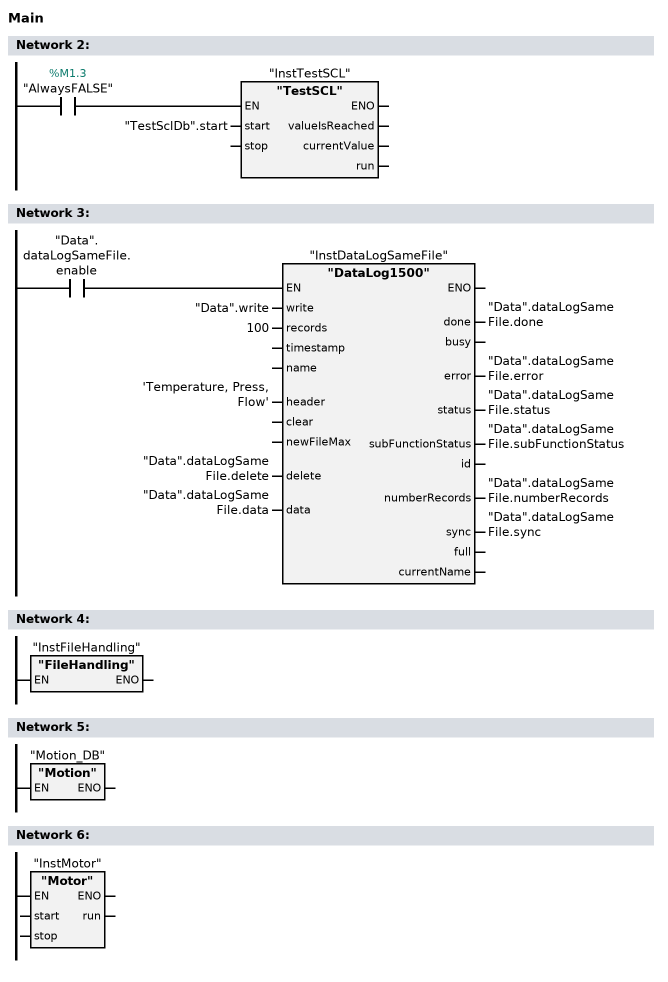
   RUNG wire#powerrail
      Contact( "AlwaysFALSE" )
      "InstTestSCL"(start := "TestSclDb".start, valueIsReached =>, currentValue =>, stop :=, run =>)
   END_RUNG
   // the same network as SCL:
   IF "AlwaysFALSE" THEN
       "InstTestSCL"(start := "TestSclDb".start);   // "TestSCL"
   END_IF;
END_REGION

REGION Network 3
   RUNG wire#powerrail
      Contact( "Data".dataLogSameFile.enable )
      "InstDataLogSameFile"(write := "Data".write, records := 100, timestamp :=, "name" :=, header := 'Temperature, Press, Flow', clear :=, newFileMax :=, delete := "Data".dataLogSameFile.delete, data := "Data".dataLogSameFile.data, done => "Data".dataLogSameFile.done, busy =>, error => "Data".dataLogSameFile.error, status => "Data".dataLogSameFile.status, subFunctionStatus => "Data".dataLogSameFile.subFunctionStatus, id =>, numberRecords => "Data".dataLogSameFile.numberRecords, sync => "Data".dataLogSameFile.sync, full =>, currentName =>)
   END_RUNG
   // the same network as SCL:
   IF "Data".dataLogSameFile.enable THEN
       "InstDataLogSameFile"(write := "Data".write,   // "DataLog1500"
                             records := 100,
                             header := 'Temperature, Press, Flow',
                             delete := "Data".dataLogSameFile.delete,
                             data := "Data".dataLogSameFile.data,
                             done => "Data".dataLogSameFile.done,
                             error => "Data".dataLogSameFile.error,
                             status => "Data".dataLogSameFile.status,
                             subFunctionStatus => "Data".dataLogSameFile.subFunctionStatus,
                             numberRecords => "Data".dataLogSameFile.numberRecords,
                             sync => "Data".dataLogSameFile.sync);
   END_IF;
END_REGION

REGION Network 4
   RUNG wire#powerrail
      "InstFileHandling"()
   END_RUNG
   // the same network as SCL:
   "InstFileHandling"();   // "FileHandling"
END_REGION

REGION Network 5
   RUNG wire#powerrail
      "Motion_DB"()
   END_RUNG
   // the same network as SCL:
   "Motion_DB"();   // "Motion"
END_REGION

REGION Network 6
   RUNG wire#powerrail
      "InstMotor"(start :=, stop :=, run =>)
   END_RUNG
   // the same network as SCL:
   "InstMotor"();   // "Motor"
END_REGION
END_ORGANIZATION_BLOCK

FUNCTION_BLOCK "TestSCL"
{ S7_Optimized_Access := 'TRUE' }
VERSION : 0.1
   VAR_INPUT 
      start : Bool;
      stop : Bool;
   END_VAR

   VAR_OUTPUT 
      valueIsReached : Bool;
      currentValue : Int;
      run : Bool;
   END_VAR

   VAR 
      instRTrigForRun {InstructionName := 'R_TRIG'; LibVersion := '1.0'} : R_TRIG;
      startRisingEdge : Bool;
   END_VAR
   VAR RETAIN
      instCounterAdd1 {InstructionName := 'CTU_INT'; LibVersion := '1.0'} : CTU_INT;
      IEC_Counter_0_Instance {InstructionName := 'CTU_INT'; LibVersion := '1.0'} : CTU_INT;
      statState { S7_SetPoint := 'True'} : DInt;
   END_VAR
   VAR 
      instRTrig {InstructionName := 'R_TRIG'; LibVersion := '1.0'} : R_TRIG;
      instLGF_FIFO : "LGF_FIFO";
      statCount { S7_SetPoint := 'True'} : Int;
      statLogFileName : String[50];
      statlogFileNameTemp : Array[0..10] of String[50];
   END_VAR

   VAR_TEMP 
      tempCount : Int;
   END_VAR

   VAR CONSTANT 
      STATE_UNDIFINED : DInt;
      STATE1 : DInt := 1;
      STATE2 : DInt := 2;
      STATE3 : DInt := 3;
      STATE4 : DInt := 4;
      STATE5 : DInt := 5;
   END_VAR


BEGIN
	IF #start THEN
	    #instRTrigForRun(CLK := TRUE,
	                     Q => #startRisingEdge);
	    
	    #instCounterAdd1(CU := TRUE,
	                     PV := 5,
	                     CV => #currentValue);
	ELSE
	    #instCounterAdd1.CU := FALSE;
	END_IF;
	
	IF #instCounterAdd1.CV = 5 THEN
	    #valueIsReached := TRUE;
	END_IF;
	
	IF #start THEN
	    IF "TestSclDb".nextStep THEN
	        #statState := #STATE1;
	    END_IF;
	END_IF;
	
	CASE #statState OF
	    #STATE1:
	        IF "TestSclDb".state1 THEN
	            #statState := #STATE2;
	        END_IF;
	        
	    #STATE2:
	        IF "TestSclDb".state2 THEN
	            #statState := #STATE3;
	        END_IF;
	        
	    #STATE3:
	        IF "TestSclDb".state3 THEN
	            #statState := #STATE4;
	        END_IF;
	END_CASE;
	
	IF "TestSclDb".cond1 = 1 THEN
	    "TestSclDb".testCond1 := TRUE;
	    #instRTrig(CLK := "TestSclDb".testCond1);
	    IF #instRTrig.Q THEN
	        "TestSclDb".result := TRUE;
	    END_IF;
	END_IF;
	
	  #instLGF_FIFO(enqueue:="Test".fifo.enqueue,
	                     dequeue:="Test".fifo.dequeue,
	                     reset:="Test".fifo.reset,
	                     clear:="Test".fifo.clear,
	                     initialItem:="Test".fifo.initialItem,
	                     item:="Test".fifo.item,
	                     buffer:="Test".fifo.buffer);
	    
	       IF #instLGF_FIFO.statElementCount = 0 THEN
	           "Test".fifo.clear := TRUE;
	       ELSE
	           "Test".fifo.clear := False;
	       END_IF;
	       
	// FOR #tempCount := 0 TO 8 DO
	//    "TestSclDb".aArray[#tempCount] := "TestSclDb".bArray[#tempCount];
	// END_FOR;
	       
	       // FOR #tempCount := 1 TO "TestSclDb".count DO
	       //     "TestSclDb".aArray[#tempCount] := "TestSclDb".bArray[#tempCount];
	       // END_FOR;
	       
	FOR #statCount := 1 TO "TestSclDb".count DO
	    "TestSclDb".aArray[#statCount] := "TestSclDb".bArray[#statCount];
	END_FOR;
	   
	"StringDb".name1 := "Test".name1;
	       
	FOR #tempCount := 1 TO 10 DO
	    "TestSclDb".string2[#tempCount] := "TestSclDb".string1[#tempCount];
	END_FOR;
	
	"TestSclDb".string3[8] := "TestSclDb".dumpString;
	#statlogFileNameTemp["TestSclDb".count] := #statLogFileName;
	
END_FUNCTION_BLOCK

FUNCTION_BLOCK "DataLog1500"
{ S7_Optimized_Access := 'TRUE' }
VERSION : 0.1
   VAR_INPUT 
      write : Bool;
      records : UDInt := 1;
      timestamp : UInt := 3;
      "name" : String := 'DataLog';
      header : String := 'Value';
      clear : Bool;
      newFileMax : USInt;
      delete : Bool;
   END_VAR

   VAR_OUTPUT 
      done { ExternalWritable := 'False'} : Bool;
      busy { ExternalWritable := 'False'} : Bool;
      error { ExternalWritable := 'False'} : Bool;
      status { ExternalWritable := 'False'} : Word := #STATUS_NO_CALL;
      subFunctionStatus { ExternalWritable := 'False'} : Word;
      id { ExternalWritable := 'False'} : DWord;
      numberRecords { ExternalWritable := 'False'} : UDInt;
      sync { ExternalWritable := 'False'} : Bool;
      full { ExternalWritable := 'False'} : Bool;
      currentName { ExternalWritable := 'False'} : String;
   END_VAR

   VAR_IN_OUT 
      data : Variant;
   END_VAR

   VAR RETAIN
      statId { ExternalAccessible := 'False'; ExternalVisible := 'False'; ExternalWritable := 'False'} : DWord;
      statNumberRecords { ExternalAccessible := 'False'; ExternalVisible := 'False'; ExternalWritable := 'False'} : UDInt;
      statSync { ExternalAccessible := 'False'; ExternalVisible := 'False'; ExternalWritable := 'False'} : Bool;
      statFull { ExternalAccessible := 'False'; ExternalVisible := 'False'; ExternalWritable := 'False'} : Bool;
      statClosed { ExternalAccessible := 'False'; ExternalVisible := 'False'; ExternalWritable := 'False'} : Bool;
      statFileNumber { ExternalAccessible := 'False'; ExternalVisible := 'False'; ExternalWritable := 'False'} : USInt;
      statName { ExternalAccessible := 'False'; ExternalVisible := 'False'; ExternalWritable := 'False'} : String;
   END_VAR
   VAR 
      statDelete { ExternalAccessible := 'False'; ExternalVisible := 'False'; ExternalWritable := 'False'} : Bool;
      statWriteOld { ExternalAccessible := 'False'; ExternalVisible := 'False'; ExternalWritable := 'False'} : Bool;
      statDeleteOld { ExternalAccessible := 'False'; ExternalVisible := 'False'; ExternalWritable := 'False'} : Bool;
      statDone { ExternalAccessible := 'False'; ExternalVisible := 'False'; ExternalWritable := 'False'} : Bool;
      statBusy { ExternalAccessible := 'False'; ExternalVisible := 'False'; ExternalWritable := 'False'} : Bool;
      statError { ExternalAccessible := 'False'; ExternalVisible := 'False'; ExternalWritable := 'False'} : Bool;
      statStatus { ExternalAccessible := 'False'; ExternalVisible := 'False'; ExternalWritable := 'False'} : Word := #STATUS_NO_CALL;
      statSubfunctionStatus { ExternalAccessible := 'False'; ExternalVisible := 'False'; ExternalWritable := 'False'} : Word;
      statFBState { ExternalAccessible := 'False'; ExternalVisible := 'False'; ExternalWritable := 'False'} : DInt := #FB_STATE_NO_PROCESSING;
      instDataLogCreate {InstructionName := 'DataLogCreate'; LibVersion := '1.0'; ExternalAccessible := 'False'; ExternalVisible := 'False'; ExternalWritable := 'False'; S7_SetPoint := 'False'} : DataLogCreate;
      instDataLogOpen {InstructionName := 'DataLogOpen'; LibVersion := '1.1'; ExternalAccessible := 'False'; ExternalVisible := 'False'; ExternalWritable := 'False'; S7_SetPoint := 'False'} : DataLogOpen;
      instDataLogWrite {InstructionName := 'DataLogWrite'; LibVersion := '1.0'; ExternalAccessible := 'False'; ExternalVisible := 'False'; ExternalWritable := 'False'; S7_SetPoint := 'False'} : DataLogWrite;
      instDataLogClear {InstructionName := 'DataLogClear'; LibVersion := '1.1'; ExternalAccessible := 'False'; ExternalVisible := 'False'; ExternalWritable := 'False'; S7_SetPoint := 'False'} : DataLogClear;
      instDataLogClose {InstructionName := 'DataLogClose'; LibVersion := '1.0'; ExternalAccessible := 'False'; ExternalVisible := 'False'; ExternalWritable := 'False'; S7_SetPoint := 'False'} : DataLogClose;
      instDataLogNewFile {InstructionName := 'DataLogNewFile'; LibVersion := '1.1'; ExternalAccessible := 'False'; ExternalVisible := 'False'; ExternalWritable := 'False'; S7_SetPoint := 'False'} : DataLogNewFile;
      instDataLogDelete {InstructionName := 'DataLogDelete'; LibVersion := '1.1'; ExternalAccessible := 'False'; ExternalVisible := 'False'; ExternalWritable := 'False'; S7_SetPoint := 'False'} : DataLogDelete;
   END_VAR

   VAR_TEMP 
      tempWrite : Bool;
      tempDelete : Bool;
      tempString : String;
      tempSize : USInt;
   END_VAR

   VAR CONSTANT 
      FB_STATE_NO_PROCESSING : DInt := 0;
      FB_STATE_CREATE : DInt := 10;
      FB_STATE_OPEN : DInt := 20;
      FB_STATE_WRITE : DInt := 30;
      FB_STATE_RECORD_OVERFLOW : DInt := 35;
      FB_STATE_CLEAR : DInt := 40;
      FB_STATE_CLOSE : DInt := 50;
      FB_STATE_FILE_OVERFLOW : DInt := 55;
      FB_STATE_NEWFILE : DInt := 60;
      FB_STATE_DELETE : DInt := 70;
      STATUS_NO_ERROR : Word := 16#0000;
      STATUS_EXECUTION_FINISHED : Word := 16#0000;
      STATUS_NO_CALL : Word := 16#7000;
      STATUS_FIRST_CALL : Word := 16#7001;
      STATUS_SUBSEQUENT_CALL : Word := 16#7002;
      STATUS_NOT_EXIST : Word := 16#8092;
      STATUS_ALREADY_EXIST : Word := 16#8093;
      STATUS_NOT_OPEN : Word := 16#80B0;
      ERR_IN_BLOCK_OPERATION : Word := 16#8001;
      ERR_PARAMETRIZATION : Word := 16#8200;
      ERR_PROCESSING_EXTERN : Word := 16#8400;
      ERR_PROCESSING_INTERN : Word := 16#8600;
      ERR_UNDEFINED_STATE : Word := 16#8600;
      ERR_DATALOGCREATE : Word := 16#8601;
      ERR_DATALOGOPEN : Word := 16#8602;
      ERR_DATALOGWRITE : Word := 16#8603;
      ERR_DATALOGCLEAR : Word := 16#8604;
      ERR_DATALOGCLOSE : Word := 16#8605;
      ERR_DATALOGNEWFILE : Word := 16#8606;
      ERR_DATALOGDELETE : Word := 16#8607;
      ERR_AREA_RESERVED : Word := 16#8800;
      ERR_USER_DEFINED_CLASSES : Word := 16#9000;
   END_VAR


BEGIN
	REGION BLOCK INFO HEADER
	  //===============================================================================
	  // Siemens AG / (c)Copyright 2020
	  //-------------------------------------------------------------------------------
	  // Title:            DataLog1200
	  // Comment/Function: A rising edge on "write" writes a record in the data log
	  //                   file "name".
	  //                   If necessary the data log file will be created or opened
	  //                   first.
	  //                   If "clear" = TRUE the data log file will be cleared before
	  //                   writing the first entry.
	  //                   If "newFileMax" > 0 a new data log file will be created to
	  //                   be written when the old is full and closed.
	  //                   This repeats until "newFileMax" is reached and than starts
	  //                   from the beginning.
	  //                   If "delete" = TRUE the data log files from "name" until
	  //                   "name_newFileMax" will be deleted.
	  //                   "write" can only be exexcuted if "delete" = FALSE.
	  //                   
	  // Author:           SIEMENS Industry Online Support (SIOS)
	  // Tested with:      CPU 1511C-1 PN V2.8
	  // Engineering:      TIA Portal V16 Update 1
	  // Restrictions:     -
	  // Requirements:     FC "Num2Name"
	  //-------------------------------------------------------------------------------
	  // Change log table:
	  // Version  | Date       | Expert in charge       | Changes applied
	  //----------|------------|------------------------|------------------------------
	  // 01.00.00 | 2020-05-14 | SIOS                   | First released version
	  //===============================================================================
	END_REGION
	
	#instDataLogCreate(RECORDS:=#records,
	                   TIMESTAMP:=#timestamp,
	                   NAME := #statName,
	                   HEADER := #header,
	                   DATA := #data,
	                   ID := #statId);
	
	#instDataLogOpen(NAME := #statName,
	                 Data := #data, // S7-1500
	                 ID := #statId);
	
	#instDataLogWrite(ID := #statId);
	
	#instDataLogClear(ID:=#statId);
	
	#instDataLogClose(ID := #statId);
	
	#instDataLogNewFile(RECORDS := #records,
	                    NAME := #statName,
	                    Data := #data, // S7-1500
	                    ID := #statId);
	
	#instDataLogDelete(NAME := #statName,
	                   ID := #statId);
	
	#tempWrite := #write; // Work with temporary value of input "write"
	#tempDelete := #delete; // Work with temporary value of input "delete"
	
	IF (#tempDelete = TRUE) AND (#statDeleteOld = FALSE) THEN // rising edge of input "delete"
	  #statFileNumber := 0;
	  #statDelete := TRUE;
	END_IF;
	
	IF (#tempDelete = FALSE) AND (#statDeleteOld = TRUE) THEN // falling edge of input "delete"
	  #statName := '';
	  #statFileNumber := 0;
	END_IF;
	
	#statDeleteOld := #tempDelete;
	
	IF #delete = false THEN
	REGION TRIGGERING
	    
	  IF (#tempWrite = TRUE) AND (#statWriteOld = FALSE) // Check if FB is triggered
	    // TODO(optional): delete next line and comment line if FB shall finish current job before new job can be started with rising edge of execute
	    AND (#statStatus = #STATUS_NO_CALL)
	  THEN // First call; initialize FB
	    #statDone := FALSE;
	    #statBusy := TRUE;
	    #statError := FALSE;
	    #statStatus := #STATUS_FIRST_CALL;
	    #statSubfunctionStatus := #STATUS_NO_ERROR;
	    IF #statFileNumber = 0 THEN
	      #statName := #name;
	    END_IF;
	    // State machine - start processing
	    #statFBState := #FB_STATE_FILE_OVERFLOW;
	    
	    // TODO: Initialize functionality: reset of variables, diagnostics, etc.
	    
	    // TODO: Initialize functionality: call subsidiary FBs with FALSE
	    //      #instFB(execute := FALSE);
	    
	    #instDataLogCreate.REQ := FALSE;
	    #instDataLogOpen.REQ := FALSE;
	    #instDataLogWrite.REQ := FALSE;
	    #instDataLogClear.REQ := FALSE;
	    #instDataLogClose.REQ := FALSE;
	    #instDataLogNewFile.REQ := FALSE;
	    #instDataLogDelete.REQ := FALSE;
	    
	  ELSIF (#statStatus = #STATUS_FIRST_CALL) THEN
	    #statStatus := #STATUS_SUBSEQUENT_CALL;
	  END_IF;
	  
	  // Edge detection 'execute' input
	  #statWriteOld := #tempWrite;
	END_REGION TRIGGERING
	
	IF (#statStatus = #STATUS_NO_CALL) THEN // Nothing to do -> End here to reduce "system load"
	  #id := #statId;
	  #numberRecords := #statNumberRecords;
	  #full := #statFull;
	  #sync := #statSync;
	  RETURN;
	END_IF;
	
	REGION STATE_MACHINE
	  CASE #statFBState OF // State machine of FB
	    #FB_STATE_NO_PROCESSING:
	      REGION NO Processing
	        // No processing active (Note: this state must always be present and left empty)
	        ;
	      END_REGION NO Processing
	      
	    #FB_STATE_FILE_OVERFLOW: // request on file overflow
	      REGION processing FILE_OVERFLOW
	        
	        IF #statClosed THEN
	          
	          "Num2Name"(nameIn := #name,
	                     number := #statFileNumber,
	                     nameOut => #statName);
	          
	          #statFBState := #FB_STATE_NEWFILE;
	          #statClosed := FALSE;
	        ELSE
	          #statFBState := #FB_STATE_RECORD_OVERFLOW;
	        END_IF;
	        
	      END_REGION processing FILE_OVERFLOW
	      
	    #FB_STATE_NEWFILE: // create new data log file
	      REGION processing NEWFILE
	        
	        #instDataLogNewFile.REQ := TRUE;
	        
	        IF #instDataLogNewFile.DONE
	        THEN
	          #statFBState := #FB_STATE_RECORD_OVERFLOW;
	          #instDataLogNewFile.REQ := FALSE;
	          #statNumberRecords := 0;
	          #statSync := TRUE;
	          #instDataLogNewFile.REQ := FALSE;
	        END_IF;
	        
	        IF #instDataLogNewFile.ERROR
	        THEN
	          CASE #instDataLogNewFile.STATUS OF
	              
	            #STATUS_ALREADY_EXIST:
	              #statId := 0;
	              #statFBState := #FB_STATE_OPEN;
	              #instDataLogNewFile.REQ := FALSE;
	              
	            ELSE
	              #statSubfunctionStatus := #instDataLogNewFile.STATUS;
	              #statStatus := #ERR_DATALOGNEWFILE;
	              
	          END_CASE;
	          
	        END_IF;
	        
	      END_REGION processing NEWFILE
	      
	    #FB_STATE_RECORD_OVERFLOW: // request on record overflow
	      REGION processing RECORD_OVERFLOW
	        
	        IF (#statNumberRecords >= #records) THEN
	          IF #clear THEN
	            #statFBState := #FB_STATE_CLEAR;
	          ELSE
	            #statFBState := #FB_STATE_WRITE;
	          END_IF;
	        ELSE
	          #statFBState := #FB_STATE_WRITE;
	        END_IF;
	        
	      END_REGION processing RECORD_OVERFLOW
	      
	    #FB_STATE_CLEAR: // clear data log
	      REGION processing CLEAR
	        
	          #instDataLogClear.REQ := TRUE;
	          
	          IF #instDataLogClear.DONE
	          THEN
	            #statFBState := #FB_STATE_WRITE;
	            #instDataLogClear.REQ := FALSE;
	          END_IF;
	          
	          IF #instDataLogClear.ERROR
	          THEN
	            
	            CASE #instDataLogClear.#STATUS OF
	                
	              #STATUS_NOT_OPEN:
	                #statFBState := #FB_STATE_OPEN;
	                #instDataLogClear.REQ := FALSE;
	                
	              #STATUS_NOT_EXIST:
	                #statFBState := #FB_STATE_CREATE;
	                #instDataLogClear.REQ := FALSE;
	                
	              ELSE
	                #statSubfunctionStatus := #instDataLogClear.STATUS;
	                #statStatus := #ERR_DATALOGCLEAR;
	                #instDataLogClear.REQ := FALSE;
	                
	            END_CASE;
	            
	          END_IF;
	        
	      END_REGION processing CLEAR
	      
	    #FB_STATE_WRITE: // write data log
	      REGION processing WRITE
	        
	        #instDataLogWrite.REQ := TRUE;
	        
	        IF #instDataLogWrite.DONE
	        THEN
	          
	          IF #statNumberRecords >= #records
	          THEN
	            #statNumberRecords := 1;
	            #statStatus := #STATUS_EXECUTION_FINISHED;
	          ELSE
	            #statNumberRecords := #statNumberRecords + 1;
	            
	            IF #statNumberRecords = #records THEN
	              
	              IF #statFileNumber < #newFileMax
	              THEN
	                #statFileNumber := #statFileNumber + 1;
	                #statFBState := #FB_STATE_CLOSE;
	              ELSE
	                #statFileNumber := 0;
	                #statId := 0;
	                #statStatus := #STATUS_EXECUTION_FINISHED;
	              END_IF;
	              
	            ELSE
	              #statStatus := #STATUS_EXECUTION_FINISHED;
	            END_IF;
	            
	          END_IF;
	          #instDataLogWrite.REQ := FALSE;
	          
	        END_IF;
	        
	        IF #instDataLogWrite.ERROR
	        THEN
	          CASE #instDataLogWrite.STATUS OF
	              
	            #STATUS_NOT_EXIST:
	              #statFBState := #FB_STATE_CREATE;
	              
	            #STATUS_NOT_OPEN:
	              #statFBState := #FB_STATE_OPEN;
	              
	            ELSE
	              #statSubfunctionStatus := #instDataLogWrite.STATUS;
	              #statStatus := #ERR_DATALOGWRITE;
	              
	          END_CASE;
	          #instDataLogWrite.REQ := FALSE;
	          
	        END_IF;
	        
	      END_REGION processing WRITE     
	      
	    #FB_STATE_CREATE: // create log
	      REGION processing CREATE
	        
	        #instDataLogCreate.REQ := TRUE;
	        
	        IF #instDataLogCreate.DONE
	        THEN
	          #statNumberRecords := 0;
	          #statSync := TRUE;
	          #statFBState := #FB_STATE_WRITE;
	          #instDataLogCreate.REQ := FALSE;
	        END_IF;
	        
	        IF #instDataLogCreate.ERROR
	        THEN
	          CASE #instDataLogCreate.STATUS OF
	              
	            #STATUS_ALREADY_EXIST:
	              #statFBState := #FB_STATE_OPEN;
	              
	            ELSE
	              #statSubfunctionStatus := #instDataLogCreate.STATUS;
	              #statStatus := #ERR_DATALOGCREATE;
	              
	          END_CASE;
	          #instDataLogCreate.REQ := FALSE;
	          
	        END_IF;
	        
	      END_REGION processing CREATE
	      
	    #FB_STATE_OPEN: // open data log
	      REGION processing OPEN
	        
	        #instDataLogOpen.REQ := TRUE;
	        
	        IF #instDataLogOpen.DONE
	        THEN
	          #statFBState := #FB_STATE_FILE_OVERFLOW;
	          #instDataLogOpen.REQ := FALSE;
	        END_IF;
	        
	        IF #instDataLogOpen.ERROR
	        THEN
	              #statSubfunctionStatus := #instDataLogOpen.STATUS;
	              #statStatus := #ERR_DATALOGOPEN;
	              #instDataLogOpen.REQ := FALSE;
	          
	        END_IF;
	        
	      END_REGION processing OPEN
	      
	    #FB_STATE_CLOSE: // close data log
	      REGION processing CLOSE
	        
	        #instDataLogClose.REQ := TRUE;
	        
	        IF #instDataLogClose.DONE
	        THEN
	          #statClosed := TRUE;
	          #statStatus := #STATUS_EXECUTION_FINISHED;
	          #instDataLogClose.REQ := FALSE;
	        END_IF;
	        
	        IF #instDataLogClose.ERROR
	        THEN
	          #statSubfunctionStatus := #instDataLogClose.STATUS;
	          #statStatus := #ERR_DATALOGCLOSE;
	          
	          #instDataLogClose.REQ := FALSE;
	        END_IF;
	        
	      END_REGION processing CLOSE
	      
	    ELSE // Undefined state in state machine reached
	      REGION undefined state
	        #statStatus := #ERR_UNDEFINED_STATE;
	      END_REGION undefined state
	  END_CASE;
	END_REGION STATE_MACHINE
	
	
	ELSE
	  // delete data log(s)
	  REGION processing DELETE
	    IF #statDelete THEN
	      IF #statFileNumber <= #newFileMax THEN
	        #statId := 0;
	        
	        IF #statFileNumber = 0 THEN
	          #statName := #name;
	        ELSE
	          "Num2Name"(nameIn := #name,
	                     number := #statFileNumber,
	                     nameOut => #statName);
	        END_IF;
	        
	        #instDataLogDelete.REQ := TRUE;
	        
	        IF #instDataLogDelete.DONE
	        THEN
	          
	          IF #statFileNumber < #newFileMax THEN
	            #statFileNumber := #statFileNumber + 1;
	          ELSE
	            #statName := '';
	            #statStatus := #STATUS_EXECUTION_FINISHED;
	            #statFileNumber := 0;
	            #statDelete := false;
	          END_IF;
	          #statNumberRecords := 0;
	          #statSync := FALSE;
	          #statFull := FALSE;
	          #instDataLogDelete.REQ := FALSE;
	        END_IF;
	        
	        IF #instDataLogDelete.ERROR
	        THEN
	          #statSubfunctionStatus := #instDataLogDelete.STATUS;
	          #statStatus := #ERR_DATALOGDELETE;
	          #statDelete := false;
	          #instDataLogDelete.REQ := FALSE;
	        END_IF;
	      END_IF;
	      
	    END_IF;
	END_REGION processing DELETE
	
	
	END_IF;
	    
	#statFull := #statNumberRecords >= #records;
	
	REGION OUTPUTS
	  // Write outputs
	  IF (#statStatus = #STATUS_EXECUTION_FINISHED) AND (#statDone = FALSE) THEN // Execution finished without errors
	    REGION execution finished
	      #statDone := TRUE;
	      #statBusy := FALSE;
	      #statError := FALSE;
	      // execution aborted --> set state no processing
	      #statFBState := #FB_STATE_NO_PROCESSING;
	    END_REGION execution finished
	    
	  ELSIF (#statStatus.%X15 = TRUE) AND (#statError = FALSE) THEN // Error occurred (#statStatus is 16#8000 to 16#FFFF)
	    REGION error occured
	      #statDone := FALSE;
	      #statBusy := FALSE;
	      #statError := TRUE;
	      // execution aborted --> set state no processing
	      #statFBState := #FB_STATE_NO_PROCESSING;
	    END_REGION error occured
	    
	  ELSIF (#tempDelete = FALSE) AND (#tempWrite = FALSE) AND ((#statDone = TRUE) OR (#statError = TRUE)) THEN // Reset outputs
	    REGION execute reseted
	      #statDone := FALSE;
	      #statBusy := FALSE;
	      #statError := FALSE;
	      #statStatus := #STATUS_NO_CALL;
	      #statSubfunctionStatus := #STATUS_NO_ERROR;
	      // TODO: Reset application specific outputs
	      // 
	    END_REGION execute reseted
	  END_IF;
	  
	  REGION Write static values to outputs
	    #done := #statDone;
	    #busy := #statBusy;
	    #error := #statError;
	    #status := #statStatus;
	    #subFunctionStatus := #statSubfunctionStatus;
	    #id := #statId;
	    #numberRecords := #statNumberRecords;
	    #full := #statFull;
	    #sync := #statSync;
	    // #currentName := #statName;
	    #currentName := CONCAT(IN1 := #statName, IN2 := '.csv');
	    // if ENO mechanism is not used / not wanted replace the following line by --> ENO := TRUE;
	    ENO := NOT #statError;
	    // TODO: Write application specific static values to outputs
	    // 
	  END_REGION Write static values TO outputs
	END_REGION OUTPUTS
END_FUNCTION_BLOCK

FUNCTION "Num2Name" : Void
{ S7_Optimized_Access := 'TRUE' }
VERSION : 0.1
   VAR_INPUT 
      nameIn : String;
      number : USInt;
   END_VAR

   VAR_OUTPUT 
      nameOut : String;
   END_VAR

   VAR_TEMP 
      tempString : String;
      tempSize : USInt;
   END_VAR

   VAR CONSTANT 
      LN_10 : Real := 2.302585;
   END_VAR


BEGIN
	REGION BLOCK INFO HEADER
	  //===============================================================================
	  // Siemens AG / (c)Copyright 2020
	  //-------------------------------------------------------------------------------
	  // Title:            Num2Name
	  // Comment/Function: "nameOut" = "<nameIn>_<number>"
	  //                   called in FB "DataLog1x00"
	  //                   
	  // Author:           SIEMENS Industry Online Support (SIOS)
	  // Tested with:      CPU 1211C V4.4 / CPU 1511C-1 PN V2.8
	  // Engineering:      TIA Portal V16 Update 1
	  // Restrictions:     -
	  // Requirements:     -
	  //-------------------------------------------------------------------------------
	  // Change log table:
	  // Version  | Date       | Expert in charge       | Changes applied
	  //----------|------------|------------------------|------------------------------
	  // 01.00.00 | 2020-05-14 | SIOS                   | First released version
	  //===============================================================================
	END_REGION
	
	#tempSize := DINT_TO_USINT(FLOOR(LN(#number) / #LN_10) + 1);
	VAL_STRG(IN := #number,
	         SIZE := #tempSize,
	         PREC := 0,
	         FORMAT := 16#0000,
	         P := 1,
	         OUT => #tempString);
	#nameOut := '';
	#nameOut := CONCAT(IN1 := #nameIn, IN2 := '_', IN3 := #tempString);
END_FUNCTION

FUNCTION_BLOCK "FileHandling"   // FB4, LAD
{ S7_Optimized_Access := 'TRUE' }
VERSION : 0.1
// stored: AutoNumber true, IsIECCheckEnabled true, IsRetainMemResEnabled false, MemoryReserve 100, SetENOAutomatically false, UDAEnableTagReadback false
   VAR
      instFileWriteC_SFB { S7_SetPoint := 'True'} : FileWriteC;
      instFileReadC_SFB { S7_SetPoint := 'True'} : FileReadC;
      instFileDelete { S7_SetPoint := 'True'} : FileDelete;
      statData { S7_SetPoint := 'True'} : Array[0..3] of Byte;
   END_VAR
BEGIN

REGION Network 1
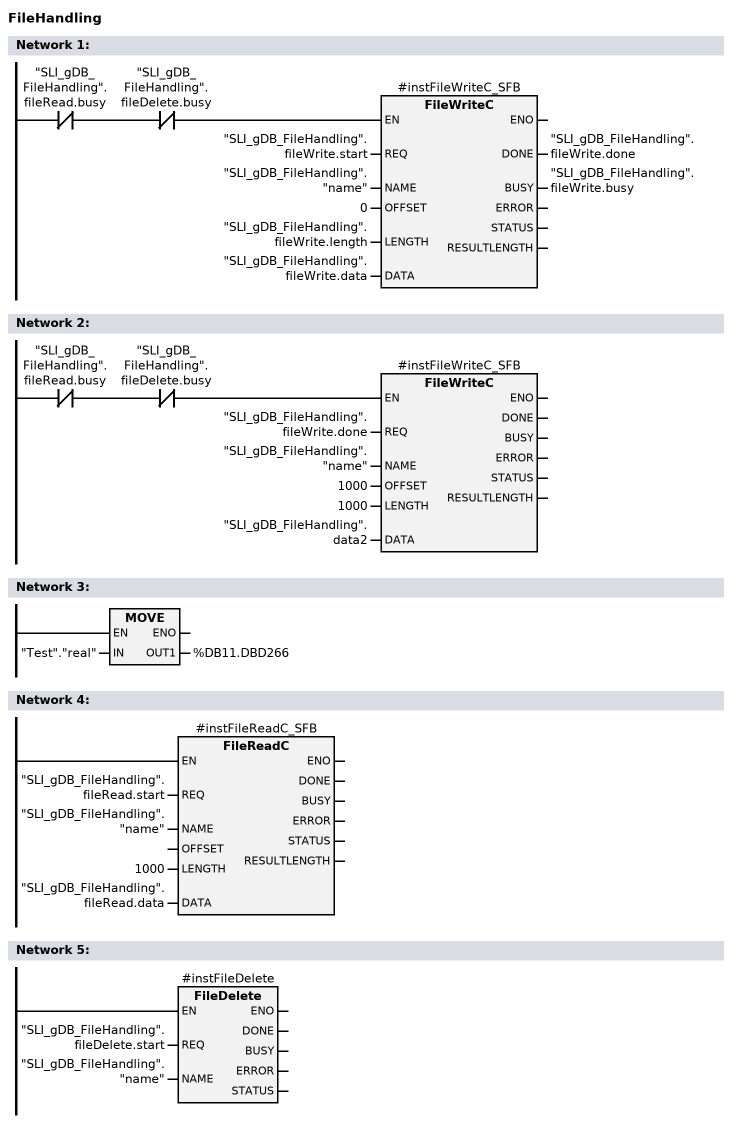
   RUNG wire#powerrail
      I_Contact( "SLI_gDB_FileHandling".fileRead.busy )
      I_Contact( "SLI_gDB_FileHandling".fileDelete.busy )
      #instFileWriteC_SFB.FileWriteC(REQ := "SLI_gDB_FileHandling".fileWrite.start, "Name" := "SLI_gDB_FileHandling"."name", Offset := 0, Length := "SLI_gDB_FileHandling".fileWrite.length, Data := "SLI_gDB_FileHandling".fileWrite.data, Done => "SLI_gDB_FileHandling".fileWrite.done, Busy => "SLI_gDB_FileHandling".fileWrite.busy, Error =>, Status =>, ResultLength =>)
   END_RUNG
   // the same network as SCL:
   IF NOT "SLI_gDB_FileHandling".fileRead.busy AND NOT "SLI_gDB_FileHandling".fileDelete.busy THEN
       #instFileWriteC_SFB(REQ := "SLI_gDB_FileHandling".fileWrite.start,   // FileWriteC
                           "Name" := "SLI_gDB_FileHandling"."name",
                           Offset := 0,
                           Length := "SLI_gDB_FileHandling".fileWrite.length,
                           Data := "SLI_gDB_FileHandling".fileWrite.data,
                           Done => "SLI_gDB_FileHandling".fileWrite.done,
                           Busy => "SLI_gDB_FileHandling".fileWrite.busy);
   END_IF;
END_REGION

REGION Network 2
   RUNG wire#powerrail
      I_Contact( "SLI_gDB_FileHandling".fileRead.busy )
      I_Contact( "SLI_gDB_FileHandling".fileDelete.busy )
      #instFileWriteC_SFB.FileWriteC(REQ := "SLI_gDB_FileHandling".fileWrite.done, "Name" := "SLI_gDB_FileHandling"."name", Offset := 1000, Length := 1000, Data := "SLI_gDB_FileHandling".data2, Done =>, Busy =>, Error =>, Status =>, ResultLength =>)
   END_RUNG
   // the same network as SCL:
   IF NOT "SLI_gDB_FileHandling".fileRead.busy AND NOT "SLI_gDB_FileHandling".fileDelete.busy THEN
       #instFileWriteC_SFB(REQ := "SLI_gDB_FileHandling".fileWrite.done,   // FileWriteC
                           "Name" := "SLI_gDB_FileHandling"."name",
                           Offset := 1000,
                           Length := 1000,
                           Data := "SLI_gDB_FileHandling".data2);
   END_IF;
END_REGION

REGION Network 3
   RUNG wire#powerrail
      Move(in := "Test"."real", out1 => %DB11.DBD266)
   END_RUNG
   // the same network as SCL:
   %DB11.DBD266 := "Test"."real";
END_REGION

REGION Network 4
   RUNG wire#powerrail
      #instFileReadC_SFB.FileReadC(REQ := "SLI_gDB_FileHandling".fileRead.start, "Name" := "SLI_gDB_FileHandling"."name", Offset :=, Length := 1000, Data := "SLI_gDB_FileHandling".fileRead.data, Done =>, Busy =>, Error =>, Status =>, ResultLength =>)
   END_RUNG
   // the same network as SCL:
   #instFileReadC_SFB(REQ := "SLI_gDB_FileHandling".fileRead.start,   // FileReadC
                      "Name" := "SLI_gDB_FileHandling"."name",
                      Length := 1000,
                      Data := "SLI_gDB_FileHandling".fileRead.data);
END_REGION

REGION Network 5
   RUNG wire#powerrail
      #instFileDelete.FileDelete(REQ := "SLI_gDB_FileHandling".fileDelete.start, "Name" := "SLI_gDB_FileHandling"."name", Done =>, Busy =>, Error =>, Status =>)
   END_RUNG
   // the same network as SCL:
   #instFileDelete(REQ := "SLI_gDB_FileHandling".fileDelete.start, "Name" := "SLI_gDB_FileHandling"."name");   // FileDelete
END_REGION
END_FUNCTION_BLOCK

FUNCTION_BLOCK "Motion"   // FB2, FBD
{ S7_Optimized_Access := 'TRUE' }
VERSION : 0.1
// stored: AutoNumber true, IsIECCheckEnabled true, IsRetainMemResEnabled false, MemoryReserve 100, SetENOAutomatically false, UDAEnableTagReadback false
   VAR
      MC_POWER_Instance { S7_SetPoint := 'True'} : MC_POWER;
      MC_RESET_Instance { S7_SetPoint := 'True'} : MC_RESET;
      MC_HOME_Instance { S7_SetPoint := 'True'} : MC_HOME;
      MC_MOVEVELOCITY_Instance { S7_SetPoint := 'True'} : MC_MOVEVELOCITY;
      MC_HALT_Instance { S7_SetPoint := 'True'} : MC_HALT;
      MC_POWER_Instance_1 { S7_SetPoint := 'True'} : MC_POWER;
      MC_RESET_Instance_1 { S7_SetPoint := 'True'} : MC_RESET;
      MC_HOME_Instance_1 { S7_SetPoint := 'True'} : MC_HOME;
      MC_MOVEVELOCITY_Instance_1 { S7_SetPoint := 'True'} : MC_MOVEVELOCITY;
      MC_HALT_Instance_1 { S7_SetPoint := 'True'} : MC_HALT;
      instMC_MOVEVELOCITY_SlsActive { S7_SetPoint := 'True'} : MC_MOVEVELOCITY;
      statSlsPtrig { S7_SetPoint := 'True'} : Bool;
   END_VAR
   VAR_TEMP   // added for the SCL form of the ladder/FBD networks
      _w1 : Bool;
   END_VAR
BEGIN

REGION Network 1
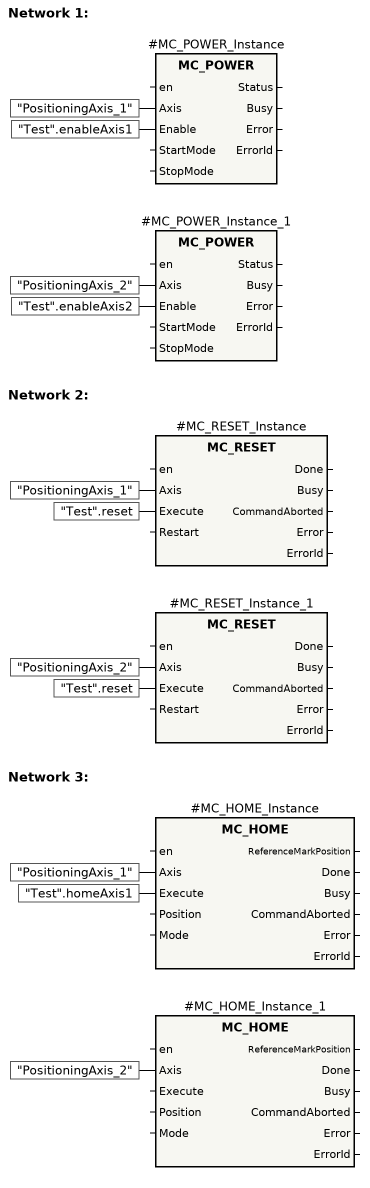
   #MC_POWER_Instance(Axis := "PositioningAxis_1", Enable := "Test".enableAxis1);   // MC_POWER
   #MC_POWER_Instance_1(Axis := "PositioningAxis_2", Enable := "Test".enableAxis2);   // MC_POWER
END_REGION

REGION Network 2
   #MC_RESET_Instance(Axis := "PositioningAxis_1", Execute := "Test".reset);   // MC_RESET
   #MC_RESET_Instance_1(Axis := "PositioningAxis_2", Execute := "Test".reset);   // MC_RESET
END_REGION

REGION Network 3
   #MC_HOME_Instance(Axis := "PositioningAxis_1", Execute := "Test".homeAxis1);   // MC_HOME
   #MC_HOME_Instance_1(Axis := "PositioningAxis_2");   // MC_HOME
END_REGION

REGION Network 4
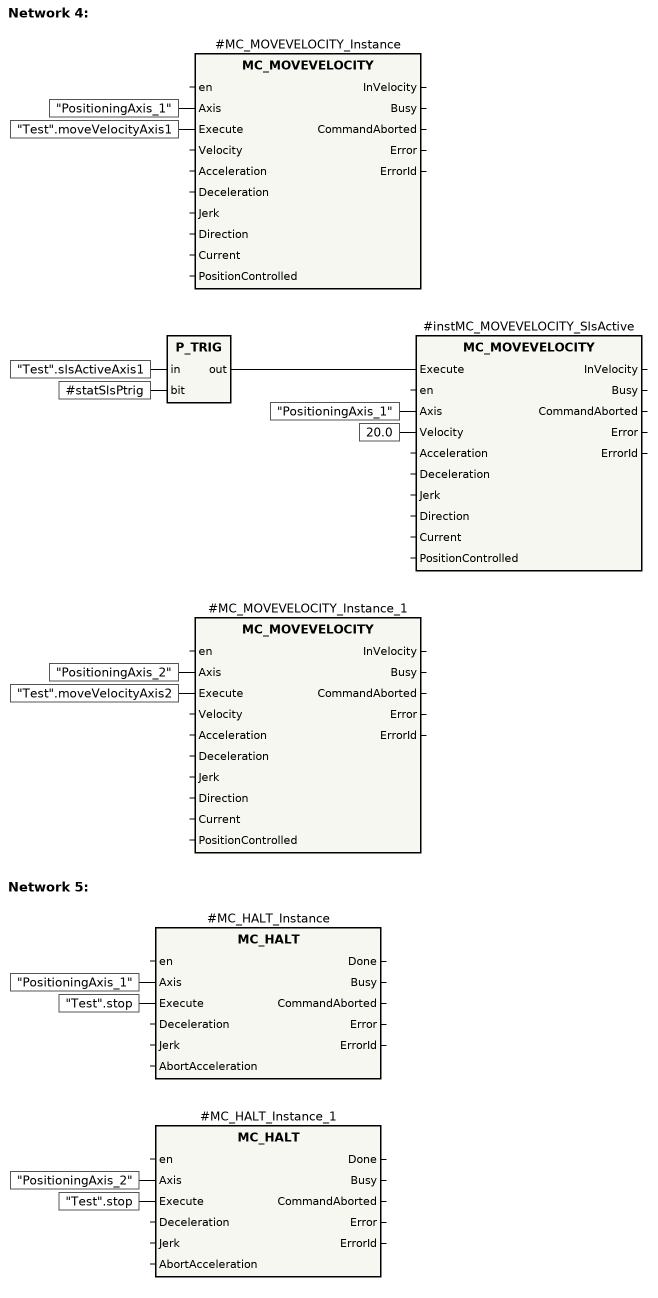
   #MC_MOVEVELOCITY_Instance(Axis := "PositioningAxis_1", Execute := "Test".moveVelocityAxis1);   // MC_MOVEVELOCITY
   #_w1 := "Test".slsActiveAxis1 AND NOT #statSlsPtrig;   // rising edge
   #statSlsPtrig := "Test".slsActiveAxis1;
   #instMC_MOVEVELOCITY_SlsActive(Execute := #_w1, Axis := "PositioningAxis_1", Velocity := 20.0);   // MC_MOVEVELOCITY
   #MC_MOVEVELOCITY_Instance_1(Axis := "PositioningAxis_2", Execute := "Test".moveVelocityAxis2);   // MC_MOVEVELOCITY
END_REGION

REGION Network 5
   #MC_HALT_Instance(Axis := "PositioningAxis_1", Execute := "Test".stop);   // MC_HALT
   #MC_HALT_Instance_1(Axis := "PositioningAxis_2", Execute := "Test".stop);   // MC_HALT
END_REGION
END_FUNCTION_BLOCK

FUNCTION_BLOCK "Motor"
{ S7_Optimized_Access := 'TRUE' }
VERSION : 0.1
   VAR_INPUT 
      start : Bool;
      stop : Bool;
   END_VAR

   VAR_OUTPUT 
      run : Bool;
   END_VAR


BEGIN
	IF #start AND NOT #stop THEN
	    #run := true;
	ELSE
	    #run := false;
	END_IF;
	
END_FUNCTION_BLOCK

ORGANIZATION_BLOCK "Rack or station failure"   // OB86, LAD, RackOrStationFailure
{ S7_Optimized_Access := 'TRUE' }
VERSION : 0.1
// stored: IsIECCheckEnabled true, SetENOAutomatically false
   VAR_INPUT
      LADDR : HW_DEVICE;   // Hardware identifier
      Event_Class : Byte;   // Event class
      Fault_ID : Byte;   // Fault identifier
   END_VAR
BEGIN
END_ORGANIZATION_BLOCK

FUNCTION_BLOCK "Main_Safety_RTG1"   // FB1, F_FBD
{ S7_Optimized_Access := 'TRUE' }
VERSION : 0.1
// stored: AutoNumber false, IsIECCheckEnabled false, UDAEnableTagReadback false
   VAR
      instACK_GL : ACK_GL;
      instLDrvSafe_SinaTlg901Control_1 : "LDrvSafe_typeSinaTlg901Control";
      instLDrvSafe_SinaTlg901Control : "LDrvSafe_SinaTlg901Control";
      instLDrvSafe_SinaTlg901Status : "LDrvSafe_SinaTlg901Status";
      instLDrvSafe_SinaSTlg30Control2 : "LDrvSafe_SinaSTlg30Control";
      instLDrvSafe_SinaSTlg30Status2 : "LDrvSafe_SinaSTlg30Status";
      instSINA_FFB : "SINA_FFB";
      instSINA_FFB1 : "SINA_FFB1";
   END_VAR
BEGIN

REGION Network 1
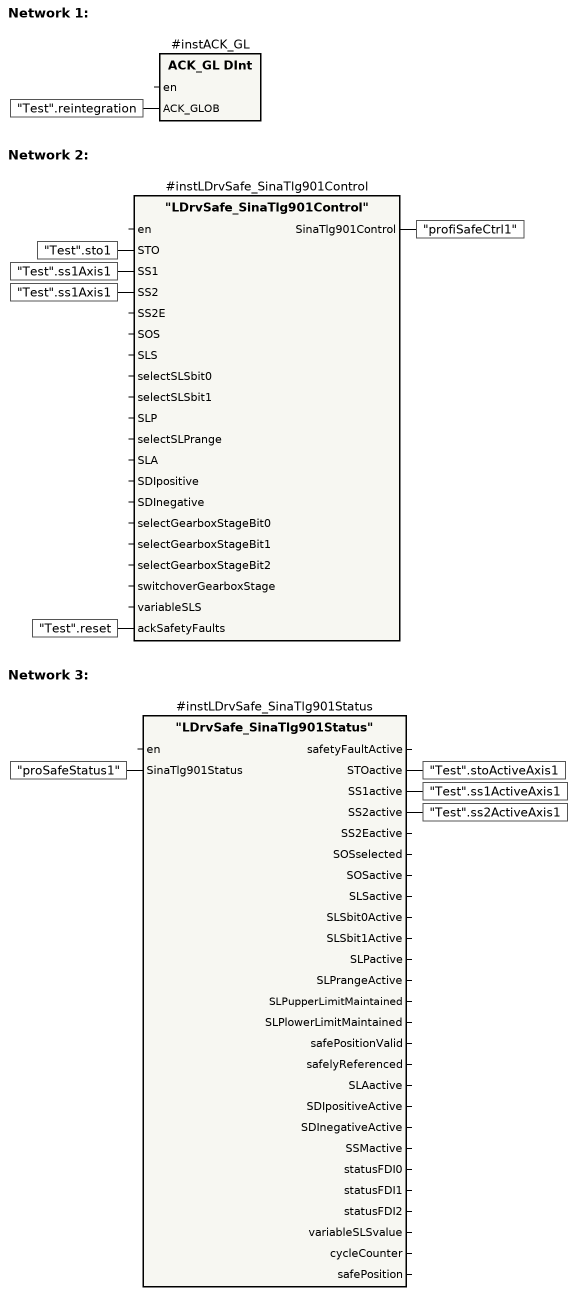
   #instACK_GL(ACK_GLOB := "Test".reintegration);   // ACK_GL
END_REGION

REGION Network 2
   #instLDrvSafe_SinaTlg901Control(STO := "Test".sto1,   // "LDrvSafe_SinaTlg901Control"
                           SS1 := "Test".ss1Axis1,
                           SS2 := "Test".ss1Axis1,
                           ackSafetyFaults := "Test".reset,
                           SinaTlg901Control => "profiSafeCtrl1");
END_REGION

REGION Network 3
   #instLDrvSafe_SinaTlg901Status(SinaTlg901Status := "proSafeStatus1",   // "LDrvSafe_SinaTlg901Status"
                           STOactive => "Test".stoActiveAxis1,
                           SS1active => "Test".ss1ActiveAxis1,
                           SS2active => "Test".ss2ActiveAxis1);
END_REGION

REGION Network 5
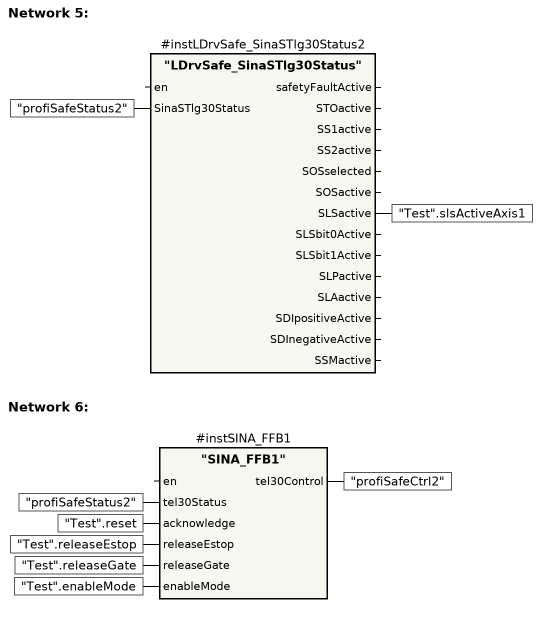
   #instLDrvSafe_SinaSTlg30Status2(SinaSTlg30Status := "profiSafeStatus2", SLSactive => "Test".slsActiveAxis1);   // "LDrvSafe_SinaSTlg30Status"
END_REGION

REGION Network 6
   #instSINA_FFB1(tel30Status := "profiSafeStatus2",   // "SINA_FFB1"
                  acknowledge := "Test".reset,
                  releaseEstop := "Test".releaseEstop,
                  releaseGate := "Test".releaseGate,
                  enableMode := "Test".enableMode,
                  tel30Control => "profiSafeCtrl2");
END_REGION
END_FUNCTION_BLOCK

FUNCTION_BLOCK "SINA_FFB1"   // FB6, F_FBD
{ S7_Optimized_Access := 'TRUE' }
VERSION : 0.1
// stored: AutoNumber true, IsIECCheckEnabled true, UDAEnableTagReadback false
   VAR_INPUT
      tel30Status : "LDrvSafe_typeSinaSTlg30Status";
      acknowledge : Bool;
      releaseEstop : Bool := true;
      releaseGate : Bool := true;
      enableMode : Bool := true;
   END_VAR
   VAR_OUTPUT
      tel30Control : "LDrvSafe_typeSinaSTlg30Control";
   END_VAR
   VAR
      statSlsTof : TOF;
      statTrue : Bool;
      statSto : Bool;
      statSs1 : Bool;
      statSs2 : Bool;
      statSos : Bool;
      statSls : Bool;
      statSlp : Bool;
      statSLA : Bool;
      statProfiSafeStatus : "LDrvSafe_typeSinaSTlg30Control";
   END_VAR
BEGIN

REGION Network 1
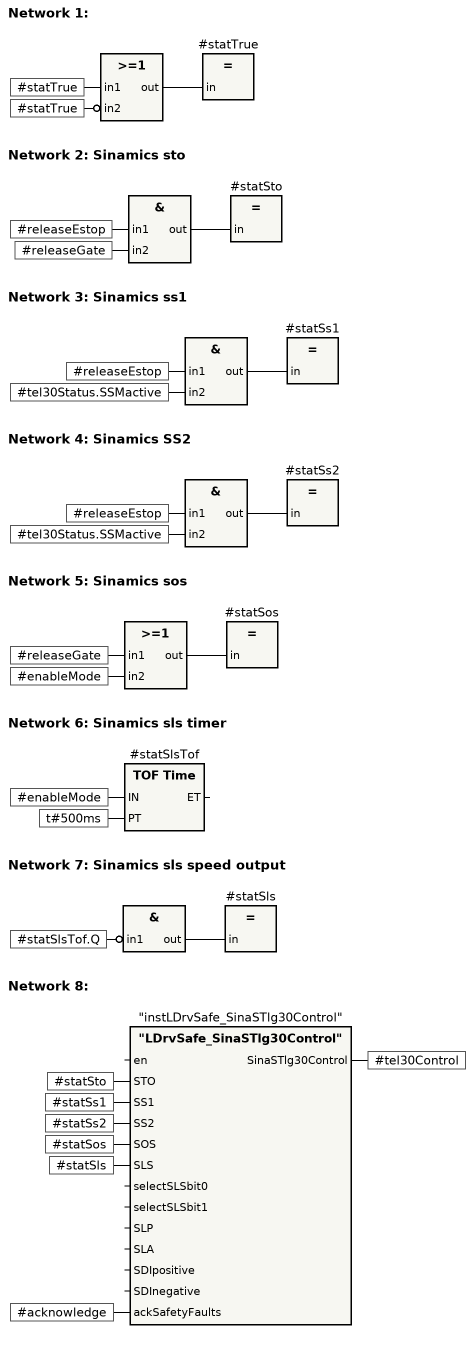
   #statTrue := #statTrue OR NOT #statTrue;
END_REGION

REGION Network 2: Sinamics sto
   #statSto := #releaseEstop AND #releaseGate;
END_REGION

REGION Network 3: Sinamics ss1
   #statSs1 := #releaseEstop AND #tel30Status.SSMactive;
END_REGION

REGION Network 4: Sinamics SS2
   #statSs2 := #releaseEstop AND #tel30Status.SSMactive;
END_REGION

REGION Network 5: Sinamics sos
   #statSos := #releaseGate OR #enableMode;
END_REGION

REGION Network 6: Sinamics sls timer
   #statSlsTof.TOF(IN := #enableMode, PT := t#500ms);
END_REGION

REGION Network 7: Sinamics sls speed output
   #statSls := NOT #statSlsTof.Q;
END_REGION

REGION Network 8
   "instLDrvSafe_SinaSTlg30Control"(STO := #statSto,   // "LDrvSafe_SinaSTlg30Control"
                           SS1 := #statSs1,
                           SS2 := #statSs2,
                           SOS := #statSos,
                           SLS := #statSls,
                           ackSafetyFaults := #acknowledge,
                           SinaSTlg30Control => #tel30Control);
END_REGION
END_FUNCTION_BLOCK

FUNCTION_BLOCK "SINA_FFB"   // FB5, F_FBD
{ S7_Optimized_Access := 'TRUE' }
VERSION : 0.1
// stored: AutoNumber true, IsIECCheckEnabled true, UDAEnableTagReadback false
   VAR_INPUT
      tel30Status : "LDrvSafe_typeSinaSTlg30Status";
      acknowledge : Bool;
      releaseEstop : Bool := true;
      releaseGate : Bool := true;
      enableMode : Bool := true;
   END_VAR
   VAR_OUTPUT
      tel30Control : "LDrvSafe_typeSinaSTlg30Control";
   END_VAR
   VAR
      statSlsTof : TOF;
      statTrue : Bool;
   END_VAR
BEGIN

REGION Network 1
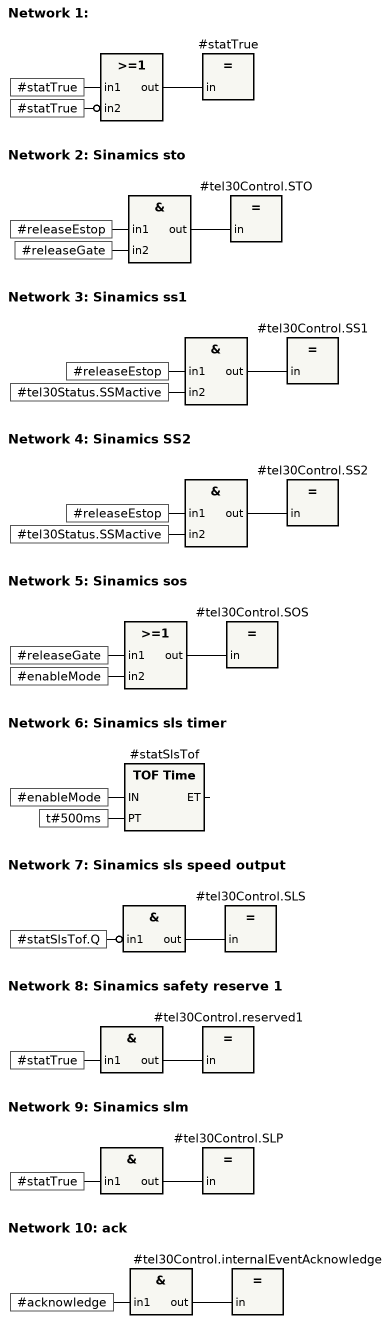
   #statTrue := #statTrue OR NOT #statTrue;
END_REGION

REGION Network 2: Sinamics sto
   #tel30Control.STO := #releaseEstop AND #releaseGate;
END_REGION

REGION Network 3: Sinamics ss1
   #tel30Control.SS1 := #releaseEstop AND #tel30Status.SSMactive;
END_REGION

REGION Network 4: Sinamics SS2
   #tel30Control.SS2 := #releaseEstop AND #tel30Status.SSMactive;
END_REGION

REGION Network 5: Sinamics sos
   #tel30Control.SOS := #releaseGate OR #enableMode;
END_REGION

REGION Network 6: Sinamics sls timer
   #statSlsTof.TOF(IN := #enableMode, PT := t#500ms);
END_REGION

REGION Network 7: Sinamics sls speed output
   #tel30Control.SLS := NOT #statSlsTof.Q;
END_REGION

REGION Network 8: Sinamics safety reserve 1
   #tel30Control.reserved1 := #statTrue;
END_REGION

REGION Network 9: Sinamics slm
   #tel30Control.SLP := #statTrue;
END_REGION

REGION Network 10: ack
   #tel30Control.internalEventAcknowledge := #acknowledge;
END_REGION

REGION Network 11: Sinamics safety reserve 2
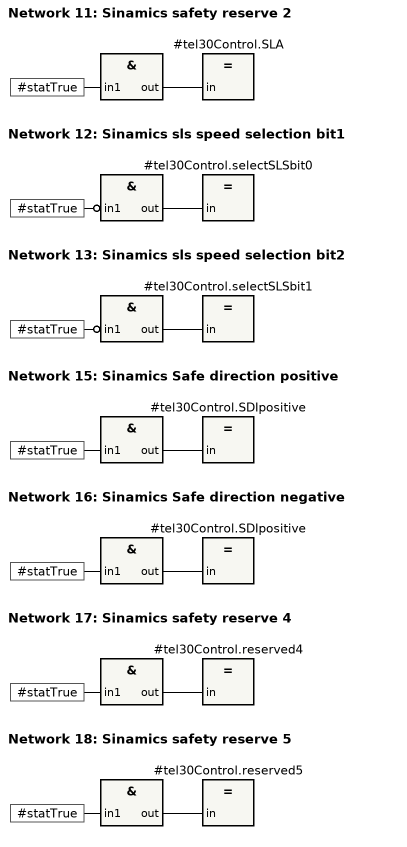
   #tel30Control.SLA := #statTrue;
END_REGION

REGION Network 12: Sinamics sls speed selection bit1
   #tel30Control.selectSLSbit0 := NOT #statTrue;
END_REGION

REGION Network 13: Sinamics sls speed selection bit2
   #tel30Control.selectSLSbit1 := NOT #statTrue;
END_REGION

REGION Network 14: Sinamics safety reserve 3
END_REGION

REGION Network 15: Sinamics Safe direction positive
   #tel30Control.SDIpositive := #statTrue;
END_REGION

REGION Network 16: Sinamics Safe direction negative
   #tel30Control.SDIpositive := #statTrue;
END_REGION

REGION Network 17: Sinamics safety reserve 4
   #tel30Control.reserved4 := #statTrue;
END_REGION

REGION Network 18: Sinamics safety reserve 5
   #tel30Control.reserved5 := #statTrue;
END_REGION
END_FUNCTION_BLOCK

FUNCTION_BLOCK "LAxisCtrl_PosAxis"
{ S7_Optimized_Access := 'TRUE' }
AUTHOR : 'tech.team.motioncontrol@siemens.com'
FAMILY : AxisCtrl
VERSION : 1.1
   VAR_INPUT 
      enable : Bool := FALSE;
      enableAxis : Bool := FALSE;
      resetAxis : Bool := FALSE;
      openBrake : Bool := FALSE;
      jogForward : Bool := FALSE;
      jogBackward : Bool := FALSE;
      moveVelocity : Bool := FALSE;
      stop : Bool := FALSE;
      fastStop : Bool := FALSE;
      torqueLimiting : Bool := FALSE;
      homing : Bool := FALSE;
      posRelative : Bool := FALSE;
      posAbsolute : Bool := FALSE;
      posSuperimposed : Bool := FALSE;
      axis {InstructionName := 'TO_PositioningAxis'; LibVersion := '5.0'} : TO_PositioningAxis;
      configuration : "LAxisCtrl_typeAxisConfig";
   END_VAR

   VAR_OUTPUT 
      valid { ExternalWritable := 'False'} : Bool := FALSE;
      busy { ExternalWritable := 'False'} : Bool := FALSE;
      error { ExternalWritable := 'False'} : Bool := FALSE;
      status { ExternalWritable := 'False'} : Word := #STATUS_NO_CALL;
      subfunctionStatus { ExternalWritable := 'False'} : Word;
      axisEnabled { ExternalWritable := 'False'} : Bool := FALSE;
      resetActive { ExternalWritable := 'False'; S7_HiddenAssignment := 'HideIfNoParamAssigned'} : Bool := FALSE;
      commandBusy { ExternalWritable := 'False'} : Bool := FALSE;
      commandDone { ExternalWritable := 'False'} : Bool := FALSE;
      commandAborted { ExternalWritable := 'False'} : Bool := FALSE;
      inVelocity { ExternalWritable := 'False'} : Bool := FALSE;
      inLimitation { ExternalWritable := 'False'; S7_HiddenAssignment := 'HideIfNoParamAssigned'} : Bool := FALSE;
      homingCommandBusy { ExternalWritable := 'False'} : Bool := FALSE;
      homingCommandDone { ExternalWritable := 'False'} : Bool := FALSE;
      homingCommandAborted { ExternalWritable := 'False'} : Bool := FALSE;
      superimposedBusy { ExternalWritable := 'False'} : Bool := FALSE;
      superimposedDone { ExternalWritable := 'False'; S7_HiddenAssignment := 'Show'} : Bool := FALSE;
      superimposedAborted { ExternalWritable := 'False'; S7_HiddenAssignment := 'Show'} : Bool := FALSE;
      inClamping { ExternalWritable := 'False'; S7_HiddenAssignment := 'HideIfNoParamAssigned'} : Bool := FALSE;
      jogSelected { ExternalWritable := 'False'; S7_HiddenAssignment := 'HideIfNoParamAssigned'} : Bool := FALSE;
      moveVelocitySelected { ExternalWritable := 'False'; S7_HiddenAssignment := 'HideIfNoParamAssigned'} : Bool := FALSE;
      stopSelected { ExternalWritable := 'False'; S7_HiddenAssignment := 'HideIfNoParamAssigned'} : Bool := FALSE;
      fastStopSelected { ExternalWritable := 'False'; S7_HiddenAssignment := 'HideIfNoParamAssigned'} : Bool := FALSE;
      torqueLimitingSelected { ExternalWritable := 'False'; S7_HiddenAssignment := 'HideIfNoParamAssigned'} : Bool := FALSE;
      homingSelected { ExternalWritable := 'False'; S7_HiddenAssignment := 'HideIfNoParamAssigned'} : Bool := FALSE;
      posRelativeSelected { ExternalWritable := 'False'; S7_HiddenAssignment := 'HideIfNoParamAssigned'} : Bool := FALSE;
      posAbsoluteSelected { ExternalWritable := 'False'; S7_HiddenAssignment := 'HideIfNoParamAssigned'} : Bool := FALSE;
      posSuperimposedSelected { ExternalWritable := 'False'; S7_HiddenAssignment := 'HideIfNoParamAssigned'} : Bool := FALSE;
      diagnostics { ExternalWritable := 'False'; S7_HiddenAssignment := 'HideIfNoParamAssigned'} : "LAxisCtrl_typeDiagnostics";
   END_VAR

